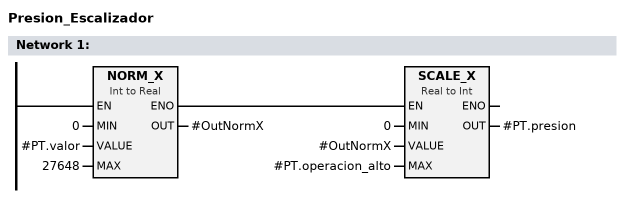
   RUNG wire#powerrail
      { S7_Templates := "[SrcType := Int, DestType := Real]"; S7_GenerateENO := "TRUE" } Normalize(min := 0, value := #PT.valor, max := 27648, out => #OutNormX)
      { S7_Templates := "[SrcType := Real, DestType := Int]"; S7_GenerateENO := "TRUE" } Scale(min := 0, value := #OutNormX, max := #PT.operacion_alto, out => #PT.presion)
   END_RUNG
   // the same network as SCL:
   // ENO of a box is taken as its EN; it also drops when the box reports an error
   #OutNormX := NORM_X(MIN := 0, VALUE := #PT.valor, MAX := 27648);
   #PT.presion := SCALE_X(MIN := 0, VALUE := #OutNormX, MAX := #PT.operacion_alto);
END_REGION
END_FUNCTION

FUNCTION "Nivel_RAD_Escalidar" : Void   // FC6, LAD
{ S7_Optimized_Access := 'TRUE' }
VERSION : 0.1
   VAR_IN_OUT
      RAD : "UDT_SENSORES_NIVEL";
   END_VAR
   VAR_TEMP
      OutNormX : Real;
      out : Int;
      Resultado_Transicion : Int;
      NivelAlto : Int;
      Resultado1 : Int;
      M1 : Real;
      M2 : Real;
   END_VAR
BEGIN

REGION Network 1
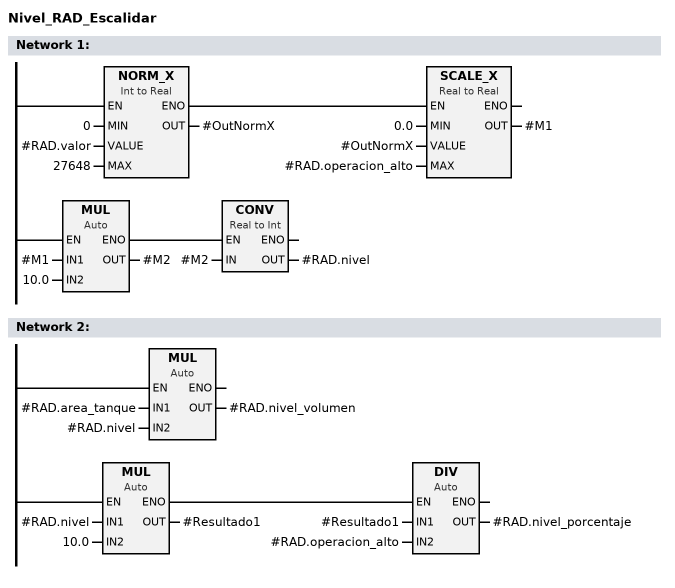
   RUNG wire#powerrail
      { S7_Templates := "[SrcType := Int, DestType := Real]"; S7_GenerateENO := "TRUE" } Normalize(min := 0, value := #RAD.valor, max := 27648, out => #OutNormX)
      { S7_Templates := "[SrcType := Real, DestType := Real]"; S7_GenerateENO := "TRUE" } Scale(min := 0.0, value := #OutNormX, max := #RAD.operacion_alto, out => #M1)
   END_RUNG
   RUNG wire#powerrail
      Mul(in1 := #M1, in2 := 10.0, out => #M2)
      { S7_Templates := "[SrcType := Real, DestType := Int]" } Convert(in := #M2, out => #RAD.nivel)
   END_RUNG
   // the same network as SCL:
   // ENO of a box is taken as its EN; it also drops when the box reports an error
   #OutNormX := NORM_X(MIN := 0, VALUE := #RAD.valor, MAX := 27648);
   #M1 := SCALE_X(MIN := 0.0, VALUE := #OutNormX, MAX := #RAD.operacion_alto);
   #M2 := #M1 * 10.0;
   #RAD.nivel := REAL_TO_INT(#M2);
END_REGION

REGION Network 2
   RUNG wire#powerrail
      Mul(in1 := #RAD.area_tanque, in2 := #RAD.nivel, out => #RAD.nivel_volumen)
   END_RUNG
   RUNG wire#powerrail
      Mul(in1 := #RAD.nivel, in2 := 10.0, out => #Resultado1)
      Div(in1 := #Resultado1, in2 := #RAD.operacion_alto, out => #RAD.nivel_porcentaje)
   END_RUNG
   // the same network as SCL:
   #RAD.nivel_volumen := #RAD.area_tanque * #RAD.nivel;
   #Resultado1 := #RAD.nivel * 10.0;
   #RAD.nivel_porcentaje := #Resultado1 / #RAD.operacion_alto;
END_REGION
END_FUNCTION

FUNCTION "Flujo_Escalizador" : Void   // FC7, LAD
{ S7_Optimized_Access := 'TRUE' }
VERSION : 0.1
   VAR_IN_OUT
      Flujo : "UDT_SENSORES_FLUJO";
   END_VAR
   VAR_TEMP
      OutNormX : Real;
      out : Int;
      Resultado_Transicion : Int;
   END_VAR
BEGIN

REGION Network 1
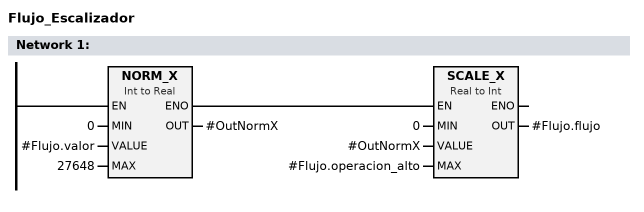
   RUNG wire#powerrail
      { S7_Templates := "[SrcType := Int, DestType := Real]"; S7_GenerateENO := "TRUE" } Normalize(min := 0, value := #Flujo.valor, max := 27648, out => #OutNormX)
      { S7_Templates := "[SrcType := Real, DestType := Int]"; S7_GenerateENO := "TRUE" } Scale(min := 0, value := #OutNormX, max := #Flujo.operacion_alto, out => #Flujo.flujo)
   END_RUNG
   // the same network as SCL:
   // ENO of a box is taken as its EN; it also drops when the box reports an error
   #OutNormX := NORM_X(MIN := 0, VALUE := #Flujo.valor, MAX := 27648);
   #Flujo.flujo := SCALE_X(MIN := 0, VALUE := #OutNormX, MAX := #Flujo.operacion_alto);
END_REGION
END_FUNCTION

ORGANIZATION_BLOCK "TransicionesINPUTOUTPUT"   // OB127, LAD, ProgramCycle
TITLE = "Main Program Sweep (Cycle)"
{ S7_Optimized_Access := 'TRUE' }
VERSION : 0.1
   VAR_INPUT
      Initial_Call : Bool;   // Initial call of this OB
      Remanence : Bool;   // =True, if remanent data are available
   END_VAR
   VAR_TEMP   // added for the SCL form of the ladder/FBD networks
      _w1 : Bool;
      _w2 : Bool;
      _w3 : Bool;
   END_VAR
BEGIN

REGION Network 1: BOMBA BC 11
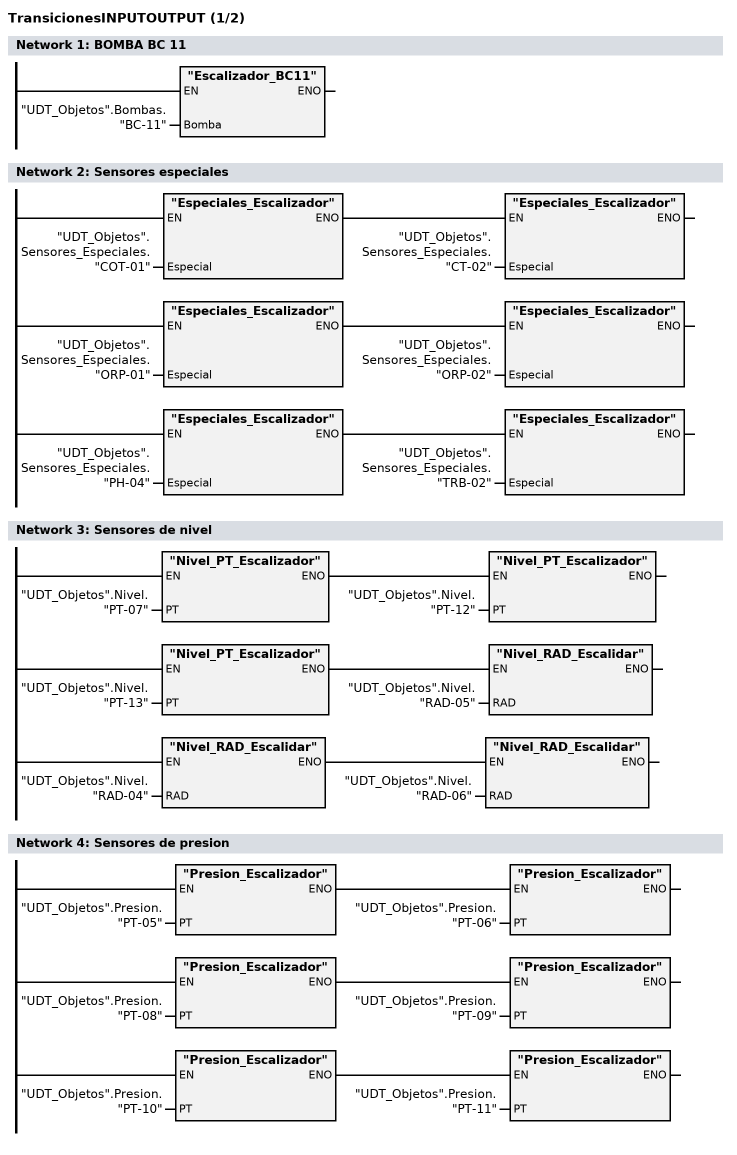
   RUNG wire#powerrail
      "Escalizador_BC11"(Bomba := "UDT_Objetos".Bombas."BC-11")
   END_RUNG
   // the same network as SCL:
   "Escalizador_BC11"(Bomba := "UDT_Objetos".Bombas."BC-11");
END_REGION

REGION Network 2: Sensores especiales
   RUNG wire#powerrail
      "Especiales_Escalizador"(Especial := "UDT_Objetos".Sensores_Especiales."COT-01")
      "Especiales_Escalizador"(Especial := "UDT_Objetos".Sensores_Especiales."CT-02")
   END_RUNG
   RUNG wire#powerrail
      "Especiales_Escalizador"(Especial := "UDT_Objetos".Sensores_Especiales."ORP-01")
      "Especiales_Escalizador"(Especial := "UDT_Objetos".Sensores_Especiales."ORP-02")
   END_RUNG
   RUNG wire#powerrail
      "Especiales_Escalizador"(Especial := "UDT_Objetos".Sensores_Especiales."PH-04")
      "Especiales_Escalizador"(Especial := "UDT_Objetos".Sensores_Especiales."TRB-02")
   END_RUNG
   // the same network as SCL:
   "Especiales_Escalizador"(Especial := "UDT_Objetos".Sensores_Especiales."COT-01", ENO => #_w1);
   IF #_w1 THEN "Especiales_Escalizador"(Especial := "UDT_Objetos".Sensores_Especiales."CT-02"); END_IF;
   "Especiales_Escalizador"(Especial := "UDT_Objetos".Sensores_Especiales."ORP-01", ENO => #_w2);
   IF #_w2 THEN "Especiales_Escalizador"(Especial := "UDT_Objetos".Sensores_Especiales."ORP-02"); END_IF;
   "Especiales_Escalizador"(Especial := "UDT_Objetos".Sensores_Especiales."PH-04", ENO => #_w3);
   IF #_w3 THEN "Especiales_Escalizador"(Especial := "UDT_Objetos".Sensores_Especiales."TRB-02"); END_IF;
END_REGION

REGION Network 3: Sensores de nivel
   RUNG wire#powerrail
      "Nivel_PT_Escalizador"(PT := "UDT_Objetos".Nivel."PT-07")
      "Nivel_PT_Escalizador"(PT := "UDT_Objetos".Nivel."PT-12")
   END_RUNG
   RUNG wire#powerrail
      "Nivel_PT_Escalizador"(PT := "UDT_Objetos".Nivel."PT-13")
      "Nivel_RAD_Escalidar"(RAD := "UDT_Objetos".Nivel."RAD-05")
   END_RUNG
   RUNG wire#powerrail
      "Nivel_RAD_Escalidar"(RAD := "UDT_Objetos".Nivel."RAD-04")
      "Nivel_RAD_Escalidar"(RAD := "UDT_Objetos".Nivel."RAD-06")
   END_RUNG
   // the same network as SCL:
   "Nivel_PT_Escalizador"(PT := "UDT_Objetos".Nivel."PT-07", ENO => #_w1);
   IF #_w1 THEN "Nivel_PT_Escalizador"(PT := "UDT_Objetos".Nivel."PT-12"); END_IF;
   "Nivel_PT_Escalizador"(PT := "UDT_Objetos".Nivel."PT-13", ENO => #_w2);
   IF #_w2 THEN "Nivel_RAD_Escalidar"(RAD := "UDT_Objetos".Nivel."RAD-05"); END_IF;
   "Nivel_RAD_Escalidar"(RAD := "UDT_Objetos".Nivel."RAD-04", ENO => #_w3);
   IF #_w3 THEN "Nivel_RAD_Escalidar"(RAD := "UDT_Objetos".Nivel."RAD-06"); END_IF;
END_REGION

REGION Network 4: Sensores de presion
   RUNG wire#powerrail
      "Presion_Escalizador"(PT := "UDT_Objetos".Presion."PT-05")
      "Presion_Escalizador"(PT := "UDT_Objetos".Presion."PT-06")
   END_RUNG
   RUNG wire#powerrail
      "Presion_Escalizador"(PT := "UDT_Objetos".Presion."PT-08")
      "Presion_Escalizador"(PT := "UDT_Objetos".Presion."PT-09")
   END_RUNG
   RUNG wire#powerrail
      "Presion_Escalizador"(PT := "UDT_Objetos".Presion."PT-10")
      "Presion_Escalizador"(PT := "UDT_Objetos".Presion."PT-11")
   END_RUNG
   // the same network as SCL:
   "Presion_Escalizador"(PT := "UDT_Objetos".Presion."PT-05", ENO => #_w1);
   IF #_w1 THEN "Presion_Escalizador"(PT := "UDT_Objetos".Presion."PT-06"); END_IF;
   "Presion_Escalizador"(PT := "UDT_Objetos".Presion."PT-08", ENO => #_w2);
   IF #_w2 THEN "Presion_Escalizador"(PT := "UDT_Objetos".Presion."PT-09"); END_IF;
   "Presion_Escalizador"(PT := "UDT_Objetos".Presion."PT-10", ENO => #_w3);
   IF #_w3 THEN "Presion_Escalizador"(PT := "UDT_Objetos".Presion."PT-11"); END_IF;
END_REGION

REGION Network 5
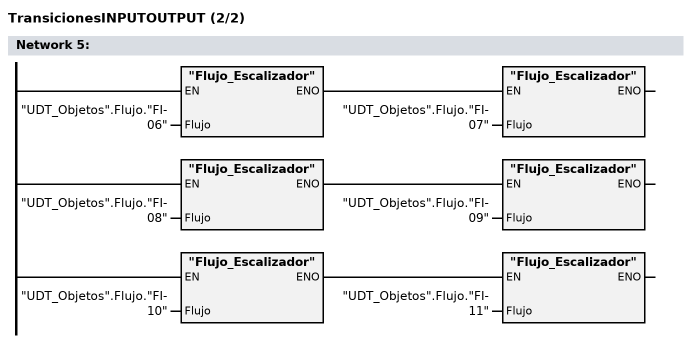
   RUNG wire#powerrail
      "Flujo_Escalizador"(Flujo := "UDT_Objetos".Flujo."FI-06")
      "Flujo_Escalizador"(Flujo := "UDT_Objetos".Flujo."FI-07")
   END_RUNG
   RUNG wire#powerrail
      "Flujo_Escalizador"(Flujo := "UDT_Objetos".Flujo."FI-08")
      "Flujo_Escalizador"(Flujo := "UDT_Objetos".Flujo."FI-09")
   END_RUNG
   RUNG wire#powerrail
      "Flujo_Escalizador"(Flujo := "UDT_Objetos".Flujo."FI-10")
      "Flujo_Escalizador"(Flujo := "UDT_Objetos".Flujo."FI-11")
   END_RUNG
   // the same network as SCL:
   "Flujo_Escalizador"(Flujo := "UDT_Objetos".Flujo."FI-06", ENO => #_w1);
   IF #_w1 THEN "Flujo_Escalizador"(Flujo := "UDT_Objetos".Flujo."FI-07"); END_IF;
   "Flujo_Escalizador"(Flujo := "UDT_Objetos".Flujo."FI-08", ENO => #_w2);
   IF #_w2 THEN "Flujo_Escalizador"(Flujo := "UDT_Objetos".Flujo."FI-09"); END_IF;
   "Flujo_Escalizador"(Flujo := "UDT_Objetos".Flujo."FI-10", ENO => #_w3);
   IF #_w3 THEN "Flujo_Escalizador"(Flujo := "UDT_Objetos".Flujo."FI-11"); END_IF;
END_REGION
END_ORGANIZATION_BLOCK

(* ===== HMI "HMI_RT_1" =====
system functions are stored by id; their names below are inferred from use
connection "HMI_Connection_1": ETHERNET, SMART_S7_1500_OMS

HMI tags "Default tag table"
   "UDT_Objetos_Bombas_BC-08_control" : Bool = PLC UDT_Objetos.Bombas.BC-08.control AT %DB1.DBX7182.0, 1 s
   "UDT_Objetos_Bombas_BC-09_control" : Bool = PLC UDT_Objetos.Bombas.BC-09.control AT %DB1.DBX7460.0, 1 s
   "UDT_Objetos_Bombas_BC-10_control" : Bool = PLC UDT_Objetos.Bombas.BC-10.control AT %DB1.DBX7738.0, 1 s
   "UDT_Objetos_Bombas_BC-11_control" : Bool = PLC UDT_Objetos.Bombas.BC-11.control AT %DB1.DBX8016.0, 1 s
   "UDT_Objetos_Bombas_BC-11_frecuencia" : Int = PLC UDT_Objetos.Bombas.BC-11.frecuencia AT %DB1.DBW8018, 1 s
   "UDT_Objetos_Bombas_BC-12_control" : Bool = PLC UDT_Objetos.Bombas.BC-12.control AT %DB1.DBX8294.0, 1 s
   "UDT_Objetos_Bombas_BC-13_control" : Bool = PLC UDT_Objetos.Bombas.BC-13.control AT %DB1.DBX8572.0, 1 s
   "UDT_Objetos_Dosificadoras_BD-AI-01_control" : Bool = PLC UDT_Objetos.Dosificadoras.BD-AI-01.control AT %DB1.DBX9938.0, 1 s
   "UDT_Objetos_Dosificadoras_BD-BIO-01_control" : Bool = PLC UDT_Objetos.Dosificadoras.BD-BIO-01.control AT %DB1.DBX10208.0, 1 s
   "UDT_Objetos_Bombas_BC-14_control" : Bool = PLC UDT_Objetos.Bombas.BC-14.control AT %DB1.DBX8850.0, 1 s
   "UDT_Objetos_Dosificadoras_BD-HIP-02_control" : Bool = PLC UDT_Objetos.Dosificadoras.BD-HIP-02.control AT %DB1.DBX10478.0, 1 s
   "UDT_Objetos_Dosificadoras_BD-HIP-01_control" : Bool = PLC UDT_Objetos.Dosificadoras.BD-HIP-01.control AT %DB1.DBX9128.0, 1 s
   "UDT_Objetos_Dosificadoras_BD-MBI-01_control" : Bool = PLC UDT_Objetos.Dosificadoras.BD-MBI-01.control AT %DB1.DBX9398.0, 1 s
   "UDT_Objetos_Dosificadoras_BD-UF-01_control" : Bool = PLC UDT_Objetos.Dosificadoras.BD-UF-01.control AT %DB1.DBX9668.0, 1 s
   "UDT_Objetos_Equipos_Especiales_BLW-01_control" : Bool = PLC UDT_Objetos.Equipos_Especiales.BLW-01.control AT %DB1.DBX25190.0, 1 s
   "UDT_Objetos_Equipos_Especiales_UV-01_control" : Bool = PLC UDT_Objetos.Equipos_Especiales.UV-01.control AT %DB1.DBX25458.0, 1 s
   "UDT_Objetos_Valvulas_VM-27_control" : Bool = PLC UDT_Objetos.Valvulas.VM-27.control AT %DB1.DBX0.0, 1 s
   "UDT_Objetos_Valvulas_VM-29_control" : Bool = PLC UDT_Objetos.Valvulas.VM-29.control AT %DB1.DBX266.0, 1 s
   "UDT_Objetos_Valvulas_VM-31_control" : Bool = PLC UDT_Objetos.Valvulas.VM-31.control AT %DB1.DBX532.0, 1 s
   "UDT_Objetos_Valvulas_VM-32_control" : Bool = PLC UDT_Objetos.Valvulas.VM-32.control AT %DB1.DBX798.0, 1 s
   "UDT_Objetos_Valvulas_VM-33_control" : Bool = PLC UDT_Objetos.Valvulas.VM-33.control AT %DB1.DBX1064.0, 1 s
   "UDT_Objetos_Valvulas_VM-34_control" : Bool = PLC UDT_Objetos.Valvulas.VM-34.control AT %DB1.DBX1330.0, 1 s
   "UDT_Objetos_Valvulas_VM-35_control" : Bool = PLC UDT_Objetos.Valvulas.VM-35.control AT %DB1.DBX1596.0, 1 s
   "UDT_Objetos_Valvulas_VM-36_control" : Bool = PLC UDT_Objetos.Valvulas.VM-36.control AT %DB1.DBX1862.0, 1 s
   "UDT_Objetos_Valvulas_VM-39_control" : Bool = PLC UDT_Objetos.Valvulas.VM-39.control AT %DB1.DBX2128.0, 1 s
   "UDT_Objetos_Valvulas_VM-40_control" : Bool = PLC UDT_Objetos.Valvulas.VM-40.control AT %DB1.DBX2394.0, 1 s
   "UDT_Objetos_Valvulas_VM-41_control" : Bool = PLC UDT_Objetos.Valvulas.VM-41.control AT %DB1.DBX2660.0, 1 s
   "UDT_Objetos_Valvulas_VM-42_control" : Bool = PLC UDT_Objetos.Valvulas.VM-42.control AT %DB1.DBX2926.0, 1 s
   "UDT_Objetos_Valvulas_VM-45_control" : Bool = PLC UDT_Objetos.Valvulas.VM-45.control AT %DB1.DBX3192.0, 1 s
   "UDT_Objetos_Valvulas_VM-46_control" : Bool = PLC UDT_Objetos.Valvulas.VM-46.control AT %DB1.DBX3458.0, 1 s
   "UDT_Objetos_Valvulas_VM-47_control" : Bool = PLC UDT_Objetos.Valvulas.VM-47.control AT %DB1.DBX3724.0, 1 s
   "UDT_Objetos_Valvulas_VM-48_control" : Bool = PLC UDT_Objetos.Valvulas.VM-48.control AT %DB1.DBX3990.0, 1 s
   "UDT_Objetos_Valvulas_VM-49_control" : Bool = PLC UDT_Objetos.Valvulas.VM-49.control AT %DB1.DBX4256.0, 1 s
   "UDT_Objetos_Valvulas_VM-50_control" : Bool = PLC UDT_Objetos.Valvulas.VM-50.control AT %DB1.DBX4522.0, 1 s
   "UDT_Objetos_Valvulas_VM-51_control" : Bool = PLC UDT_Objetos.Valvulas.VM-51.control AT %DB1.DBX4788.0, 1 s
   "UDT_Objetos_Valvulas_VM-52_control" : Bool = PLC UDT_Objetos.Valvulas.VM-52.control AT %DB1.DBX5054.0, 1 s
   "UDT_Objetos_Valvulas_VM-53_control" : Bool = PLC UDT_Objetos.Valvulas.VM-53.control AT %DB1.DBX5320.0, 1 s
   "UDT_Objetos_Valvulas_VM-56_control" : Bool = PLC UDT_Objetos.Valvulas.VM-56.control AT %DB1.DBX5586.0, 1 s
   "UDT_Objetos_Valvulas_VM-57_control" : Bool = PLC UDT_Objetos.Valvulas.VM-57.control AT %DB1.DBX5852.0, 1 s
   "UDT_Objetos_Valvulas_VM-58_control" : Bool = PLC UDT_Objetos.Valvulas.VM-58.control AT %DB1.DBX6118.0, 1 s
   "UDT_Objetos_Valvulas_VM-61_control" : Bool = PLC UDT_Objetos.Valvulas.VM-61.control AT %DB1.DBX6384.0, 1 s
   "UDT_Objetos_Valvulas_VM-62_control" : Bool = PLC UDT_Objetos.Valvulas.VM-62.control AT %DB1.DBX6650.0, 1 s
   "UDT_Objetos_Valvulas_VM-63_control" : Bool = PLC UDT_Objetos.Valvulas.VM-63.control AT %DB1.DBX6916.0, 1 s
   "UDT_Objetos_Valvulas_VM-27_estado" : Int = PLC UDT_Objetos.Valvulas.VM-27.estado AT %DB1.DBW2, 1 s
   "UDT_Objetos_Valvulas_VM-29_estado" : Int = PLC UDT_Objetos.Valvulas.VM-29.estado AT %DB1.DBW268, 1 s
   "UDT_Objetos_Valvulas_VM-31_estado" : Int = PLC UDT_Objetos.Valvulas.VM-31.estado AT %DB1.DBW534, 1 s
   "UDT_Objetos_Valvulas_VM-32_estado" : Int = PLC UDT_Objetos.Valvulas.VM-32.estado AT %DB1.DBW800, 1 s
   "UDT_Objetos_Valvulas_VM-33_estado" : Int = PLC UDT_Objetos.Valvulas.VM-33.estado AT %DB1.DBW1066, 1 s
   "UDT_Objetos_Valvulas_VM-34_estado" : Int = PLC UDT_Objetos.Valvulas.VM-34.estado AT %DB1.DBW1332, 1 s
   "UDT_Objetos_Valvulas_VM-35_estado" : Int = PLC UDT_Objetos.Valvulas.VM-35.estado AT %DB1.DBW1598, 1 s
   "UDT_Objetos_Valvulas_VM-36_estado" : Int = PLC UDT_Objetos.Valvulas.VM-36.estado AT %DB1.DBW1864, 1 s
   "UDT_Objetos_Valvulas_VM-39_estado" : Int = PLC UDT_Objetos.Valvulas.VM-39.estado AT %DB1.DBW2130, 1 s
   "UDT_Objetos_Valvulas_VM-40_estado" : Int = PLC UDT_Objetos.Valvulas.VM-40.estado AT %DB1.DBW2396, 1 s
   "UDT_Objetos_Valvulas_VM-41_estado" : Int = PLC UDT_Objetos.Valvulas.VM-41.estado AT %DB1.DBW2662, 1 s
   "UDT_Objetos_Valvulas_VM-42_estado" : Int = PLC UDT_Objetos.Valvulas.VM-42.estado AT %DB1.DBW2928, 1 s
   "UDT_Objetos_Valvulas_VM-45_estado" : Int = PLC UDT_Objetos.Valvulas.VM-45.estado AT %DB1.DBW3194, 1 s
   "UDT_Objetos_Valvulas_VM-46_estado" : Int = PLC UDT_Objetos.Valvulas.VM-46.estado AT %DB1.DBW3460, 1 s
   "UDT_Objetos_Valvulas_VM-47_estado" : Int = PLC UDT_Objetos.Valvulas.VM-47.estado AT %DB1.DBW3726, 1 s
   "UDT_Objetos_Valvulas_VM-48_estado" : Int = PLC UDT_Objetos.Valvulas.VM-48.estado AT %DB1.DBW3992, 1 s
   "UDT_Objetos_Valvulas_VM-49_estado" : Int = PLC UDT_Objetos.Valvulas.VM-49.estado AT %DB1.DBW4258, 1 s
   "UDT_Objetos_Valvulas_VM-50_estado" : Int = PLC UDT_Objetos.Valvulas.VM-50.estado AT %DB1.DBW4524, 1 s
   "UDT_Objetos_Valvulas_VM-51_estado" : Int = PLC UDT_Objetos.Valvulas.VM-51.estado AT %DB1.DBW4790, 1 s
   "UDT_Objetos_Valvulas_VM-52_estado" : Int = PLC UDT_Objetos.Valvulas.VM-52.estado AT %DB1.DBW5056, 1 s
   "UDT_Objetos_Valvulas_VM-53_estado" : Int = PLC UDT_Objetos.Valvulas.VM-53.estado AT %DB1.DBW5322, 1 s
   "UDT_Objetos_Valvulas_VM-56_estado" : Int = PLC UDT_Objetos.Valvulas.VM-56.estado AT %DB1.DBW5588, 1 s
   "UDT_Objetos_Valvulas_VM-57_estado" : Int = PLC UDT_Objetos.Valvulas.VM-57.estado AT %DB1.DBW5854, 1 s
   "UDT_Objetos_Valvulas_VM-58_estado" : Int = PLC UDT_Objetos.Valvulas.VM-58.estado AT %DB1.DBW6120, 1 s
   "UDT_Objetos_Valvulas_VM-61_estado" : Int = PLC UDT_Objetos.Valvulas.VM-61.estado AT %DB1.DBW6386, 1 s
   "UDT_Objetos_Valvulas_VM-62_estado" : Int = PLC UDT_Objetos.Valvulas.VM-62.estado AT %DB1.DBW6652, 1 s
   "UDT_Objetos_Valvulas_VM-63_estado" : Int = PLC UDT_Objetos.Valvulas.VM-63.estado AT %DB1.DBW6918, 1 s
   "UDT_Objetos_Bombas_BC-08_feedback" : Bool = PLC UDT_Objetos.Bombas.BC-08.feedback AT %DB1.DBX7186.0, 1 s
   "UDT_Objetos_Bombas_BC-08_estado" : Int = PLC UDT_Objetos.Bombas.BC-08.estado AT %DB1.DBW7192, 1 s
   "UDT_Objetos_Bombas_BC-09_estado" : Int = PLC UDT_Objetos.Bombas.BC-09.estado AT %DB1.DBW7470, 1 s
   "UDT_Objetos_Bombas_BC-10_estado" : Int = PLC UDT_Objetos.Bombas.BC-10.estado AT %DB1.DBW7748, 1 s
   "UDT_Objetos_Bombas_BC-11_estado" : Int = PLC UDT_Objetos.Bombas.BC-11.estado AT %DB1.DBW8026, 1 s
   "UDT_Objetos_Bombas_BC-12_estado" : Int = PLC UDT_Objetos.Bombas.BC-12.estado AT %DB1.DBW8304, 1 s
   "UDT_Objetos_Bombas_BC-13_estado" : Int = PLC UDT_Objetos.Bombas.BC-13.estado AT %DB1.DBW8582, 1 s
   "UDT_Objetos_Bombas_BC-14_estado" : Int = PLC UDT_Objetos.Bombas.BC-14.estado AT %DB1.DBW8860, 1 s
   "UDT_Objetos_Dosificadoras_BD-AI-01_estado" : Int = PLC UDT_Objetos.Dosificadoras.BD-AI-01.estado AT %DB1.DBW9940, 1 s
   "UDT_Objetos_Dosificadoras_BD-BIO-01_estado" : Int = PLC UDT_Objetos.Dosificadoras.BD-BIO-01.estado AT %DB1.DBW10210, 1 s
   "UDT_Objetos_Dosificadoras_BD-HIP-01_estado" : Int = PLC UDT_Objetos.Dosificadoras.BD-HIP-01.estado AT %DB1.DBW9130, 1 s
   "UDT_Objetos_Dosificadoras_BD-HIP-02_estado" : Int = PLC UDT_Objetos.Dosificadoras.BD-HIP-02.estado AT %DB1.DBW10480, 1 s
   "UDT_Objetos_Dosificadoras_BD-MBI-01_estado" : Int = PLC UDT_Objetos.Dosificadoras.BD-MBI-01.estado AT %DB1.DBW9400, 1 s
   "UDT_Objetos_Dosificadoras_BD-UF-01_estado" : Int = PLC UDT_Objetos.Dosificadoras.BD-UF-01.estado AT %DB1.DBW9670, 1 s
   "UDT_Objetos_Equipos_Especiales_BLW-01_estado" : Int = PLC UDT_Objetos.Equipos_Especiales.BLW-01.estado AT %DB1.DBW25194, 1 s
   "UDT_Objetos_Equipos_Especiales_UV-01_estado" : Int = PLC UDT_Objetos.Equipos_Especiales.UV-01.estado AT %DB1.DBW25462, 1 s
   "Solito" : Word = PLC Solito AT %MW2, 1 s
   "UDT_Objetos_Sensores_Especiales_COT-01_operacion_bajo" : Int = PLC UDT_Objetos.Sensores_Especiales.COT-01.operacion_bajo AT %DB1.DBW24920, 1 s
   "UDT_Objetos_Sensores_Especiales_COT-01_operacion_alto" : Int = PLC UDT_Objetos.Sensores_Especiales.COT-01.operacion_alto AT %DB1.DBW24918, 1 s
   "UDT_Objetos_Sensores_Especiales_COT-01_trabajo_alto" : Int = PLC UDT_Objetos.Sensores_Especiales.COT-01.trabajo_alto AT %DB1.DBW24924, 1 s
   "UDT_Objetos_Sensores_Especiales_CT-02_operacion_bajo" : Int = PLC UDT_Objetos.Sensores_Especiales.CT-02.operacion_bajo AT %DB1.DBW24390, 1 s
   "UDT_Objetos_Sensores_Especiales_CT-02_operacion_alto" : Int = PLC UDT_Objetos.Sensores_Especiales.CT-02.operacion_alto AT %DB1.DBW24388, 1 s
   "UDT_Objetos_Sensores_Especiales_CT-02_trabajo_alto" : Int = PLC UDT_Objetos.Sensores_Especiales.CT-02.trabajo_alto AT %DB1.DBW24394, 1 s
   "UDT_Objetos_Sensores_Especiales_CT-02_trabajo_bajo" : Int = PLC UDT_Objetos.Sensores_Especiales.CT-02.trabajo_bajo AT %DB1.DBW24396, 1 s
   "UDT_Objetos_Sensores_Especiales_ORP-01_operacion_bajo" : Int = PLC UDT_Objetos.Sensores_Especiales.ORP-01.operacion_bajo AT %DB1.DBW22800, 1 s
   "UDT_Objetos_Sensores_Especiales_ORP-01_operacion_alto" : Int = PLC UDT_Objetos.Sensores_Especiales.ORP-01.operacion_alto AT %DB1.DBW22798, 1 s
   "UDT_Objetos_Sensores_Especiales_ORP-01_trabajo_alto" : Int = PLC UDT_Objetos.Sensores_Especiales.ORP-01.trabajo_alto AT %DB1.DBW22804, 1 s
   "UDT_Objetos_Sensores_Especiales_ORP-01_trabajo_bajo" : Int = PLC UDT_Objetos.Sensores_Especiales.ORP-01.trabajo_bajo AT %DB1.DBW22806, 1 s
   "UDT_Objetos_Sensores_Especiales_ORP-02_operacion_bajo" : Int = PLC UDT_Objetos.Sensores_Especiales.ORP-02.operacion_bajo AT %DB1.DBW23330, 1 s
   "UDT_Objetos_Sensores_Especiales_ORP-02_operacion_alto" : Int = PLC UDT_Objetos.Sensores_Especiales.ORP-02.operacion_alto AT %DB1.DBW23328, 1 s
   "UDT_Objetos_Sensores_Especiales_ORP-02_trabajo_alto" : Int = PLC UDT_Objetos.Sensores_Especiales.ORP-02.trabajo_alto AT %DB1.DBW23334, 1 s
   "UDT_Objetos_Sensores_Especiales_ORP-02_trabajo_bajo" : Int = PLC UDT_Objetos.Sensores_Especiales.ORP-02.trabajo_bajo AT %DB1.DBW23336, 1 s
   "UDT_Objetos_Sensores_Especiales_PH-04_operacion_bajo" : Int = PLC UDT_Objetos.Sensores_Especiales.PH-04.operacion_bajo AT %DB1.DBW23860, 1 s
   "UDT_Objetos_Sensores_Especiales_TRB-02_operacion_bajo" : Int = PLC UDT_Objetos.Sensores_Especiales.TRB-02.operacion_bajo AT %DB1.DBW22270, 1 s
   "UDT_Objetos_Sensores_Especiales_TRB-02_operacion_alto" : Int = PLC UDT_Objetos.Sensores_Especiales.TRB-02.operacion_alto AT %DB1.DBW22268, 1 s
   "UDT_Objetos_Sensores_Especiales_TRB-02_trabajo_alto" : Int = PLC UDT_Objetos.Sensores_Especiales.TRB-02.trabajo_alto AT %DB1.DBW22274, 1 s
   "UDT_Objetos_Sensores_Especiales_TRB-02_trabajo_bajo" : Int = PLC UDT_Objetos.Sensores_Especiales.TRB-02.trabajo_bajo AT %DB1.DBW22276, 1 s
   "UDT_Objetos_Flujo_FI-06_operacion_bajo" : Int = PLC UDT_Objetos.Flujo.FI-06.operacion_bajo AT %DB1.DBW19330, 1 s
   "UDT_Objetos_Flujo_FI-06_operacion_alto" : Int = PLC UDT_Objetos.Flujo.FI-06.operacion_alto AT %DB1.DBW19328, 1 s
   "UDT_Objetos_Flujo_FI-06_trabajo_alto" : Int = PLC UDT_Objetos.Flujo.FI-06.trabajo_alto AT %DB1.DBW19332, 1 s
   "UDT_Objetos_Flujo_FI-06_trabajo_bajo" : Int = PLC UDT_Objetos.Flujo.FI-06.trabajo_bajo AT %DB1.DBW19334, 1 s
   "UDT_Objetos_Flujo_FI-07_operacion_bajo" : Int = PLC UDT_Objetos.Flujo.FI-07.operacion_bajo AT %DB1.DBW19864, 1 s
   "UDT_Objetos_Flujo_FI-07_operacion_alto" : Int = PLC UDT_Objetos.Flujo.FI-07.operacion_alto AT %DB1.DBW19862, 1 s
   "UDT_Objetos_Flujo_FI-07_trabajo_alto" : Int = PLC UDT_Objetos.Flujo.FI-07.trabajo_alto AT %DB1.DBW19866, 1 s
   "UDT_Objetos_Flujo_FI-07_trabajo_bajo" : Int = PLC UDT_Objetos.Flujo.FI-07.trabajo_bajo AT %DB1.DBW19868, 1 s
   "UDT_Objetos_Flujo_FI-08_operacion_bajo" : Int = PLC UDT_Objetos.Flujo.FI-08.operacion_bajo AT %DB1.DBW20398, 1 s
   "UDT_Objetos_Flujo_FI-08_operacion_alto" : Int = PLC UDT_Objetos.Flujo.FI-08.operacion_alto AT %DB1.DBW20396, 1 s
   "UDT_Objetos_Flujo_FI-08_trabajo_alto" : Int = PLC UDT_Objetos.Flujo.FI-08.trabajo_alto AT %DB1.DBW20400, 1 s
   "UDT_Objetos_Flujo_FI-08_trabajo_bajo" : Int = PLC UDT_Objetos.Flujo.FI-08.trabajo_bajo AT %DB1.DBW20402, 1 s
   "UDT_Objetos_Flujo_FI-09_operacion_bajo" : Int = PLC UDT_Objetos.Flujo.FI-09.operacion_bajo AT %DB1.DBW20932, 1 s
   "UDT_Objetos_Flujo_FI-09_operacion_alto" : Int = PLC UDT_Objetos.Flujo.FI-09.operacion_alto AT %DB1.DBW20930, 1 s
   "UDT_Objetos_Flujo_FI-09_trabajo_alto" : Int = PLC UDT_Objetos.Flujo.FI-09.trabajo_alto AT %DB1.DBW20934, 1 s
   "UDT_Objetos_Flujo_FI-09_trabajo_bajo" : Int = PLC UDT_Objetos.Flujo.FI-09.trabajo_bajo AT %DB1.DBW20936, 1 s
   "UDT_Objetos_Flujo_FI-11_operacion_alto" : Int = PLC UDT_Objetos.Flujo.FI-11.operacion_alto AT %DB1.DBW21998, 1 s
   "UDT_Objetos_Flujo_FI-11_trabajo_alto" : Int = PLC UDT_Objetos.Flujo.FI-11.trabajo_alto AT %DB1.DBW22002, 1 s
   "UDT_Objetos_Flujo_FI-11_trabajo_bajo" : Int = PLC UDT_Objetos.Flujo.FI-11.trabajo_bajo AT %DB1.DBW22004, 1 s
   "UDT_Objetos_Nivel_RAD-04_rango_alto" : Int = PLC UDT_Objetos.Nivel.RAD-04.operacion_alto AT %DB1.DBW11274, 1 s
   "UDT_Objetos_Nivel_RAD-05_rango_alto" : Int = PLC UDT_Objetos.Nivel.RAD-05.operacion_alto AT %DB1.DBW11816, 1 s
   "UDT_Objetos_Nivel_RAD-06_rango_alto" : Int = PLC UDT_Objetos.Nivel.RAD-06.operacion_alto AT %DB1.DBW12358, 1 s
   "UDT_Objetos_Nivel_RAD-04_rango_bajo" : Int = PLC UDT_Objetos.Nivel.RAD-04.rango_bajo AT %DB1.DBW11276, 1 s
   "UDT_Objetos_Nivel_RAD-04_rango_medio_bajo" : Int = PLC UDT_Objetos.Nivel.RAD-04.rango_medio_bajo AT %DB1.DBW11278, 1 s
   "UDT_Objetos_Nivel_RAD-04_rango_medio_alto" : Int = PLC UDT_Objetos.Nivel.RAD-04.rango_medio_alto AT %DB1.DBW11280, 1 s
   "UDT_Objetos_Nivel_RAD-04_rango_alto(1)" : Int = PLC UDT_Objetos.Nivel.RAD-04.rango_alto AT %DB1.DBW11282, 1 s
   "UDT_Objetos_Nivel_RAD-05_rango_bajo" : Int = PLC UDT_Objetos.Nivel.RAD-05.rango_bajo AT %DB1.DBW11818, 1 s
   "UDT_Objetos_Nivel_RAD-05_rango_medio_bajo" : Int = PLC UDT_Objetos.Nivel.RAD-05.rango_medio_bajo AT %DB1.DBW11820, 1 s
   "UDT_Objetos_Nivel_RAD-05_rango_medio_alto" : Int = PLC UDT_Objetos.Nivel.RAD-05.rango_medio_alto AT %DB1.DBW11822, 1 s
   "UDT_Objetos_Nivel_RAD-05_rango_alto(1)" : Int = PLC UDT_Objetos.Nivel.RAD-05.rango_alto AT %DB1.DBW11824, 1 s
   "UDT_Objetos_Nivel_RAD-06_rango_bajo" : Int = PLC UDT_Objetos.Nivel.RAD-06.rango_bajo AT %DB1.DBW12360, 1 s
   "UDT_Objetos_Nivel_RAD-06_rango_medio_bajo" : Int = PLC UDT_Objetos.Nivel.RAD-06.rango_medio_bajo AT %DB1.DBW12362, 1 s
   "UDT_Objetos_Nivel_RAD-06_rango_medio_alto" : Int = PLC UDT_Objetos.Nivel.RAD-06.rango_medio_alto AT %DB1.DBW12364, 1 s
   "UDT_Objetos_Nivel_RAD-06_rango_alto(1)" : Int = PLC UDT_Objetos.Nivel.RAD-06.rango_alto AT %DB1.DBW12366, 1 s
   "UDT_Objetos_Presion_PT-05_operacion_bajo" : Int = PLC UDT_Objetos.Presion.PT-05.operacion_bajo AT %DB1.DBW16148, 1 s
   "UDT_Objetos_Presion_PT-05_operacion_alto" : Int = PLC UDT_Objetos.Presion.PT-05.operacion_alto AT %DB1.DBW16146, 1 s
   "UDT_Objetos_Presion_PT-05_trabajo_bajo" : Int = PLC UDT_Objetos.Presion.PT-05.trabajo_bajo AT %DB1.DBW16152, 1 s
   "UDT_Objetos_Presion_PT-05_trabajo_alto" : Int = PLC UDT_Objetos.Presion.PT-05.trabajo_alto AT %DB1.DBW16150, 1 s
   "UDT_Objetos_Presion_PT-06_operacion_bajo" : Int = PLC UDT_Objetos.Presion.PT-06.operacion_bajo AT %DB1.DBW16678, 1 s
   "UDT_Objetos_Presion_PT-06_operacion_alto" : Int = PLC UDT_Objetos.Presion.PT-06.operacion_alto AT %DB1.DBW16676, 1 s
   "UDT_Objetos_Presion_PT-06_trabajo_bajo" : Int = PLC UDT_Objetos.Presion.PT-06.trabajo_bajo AT %DB1.DBW16682, 1 s
   "UDT_Objetos_Presion_PT-06_trabajo_alto" : Int = PLC UDT_Objetos.Presion.PT-06.trabajo_alto AT %DB1.DBW16680, 1 s
   "UDT_Objetos_Presion_PT-08_operacion_bajo" : Int = PLC UDT_Objetos.Presion.PT-08.operacion_bajo AT %DB1.DBW17208, 1 s
   "UDT_Objetos_Presion_PT-08_operacion_alto" : Int = PLC UDT_Objetos.Presion.PT-08.operacion_alto AT %DB1.DBW17206, 1 s
   "UDT_Objetos_Presion_PT-08_trabajo_bajo" : Int = PLC UDT_Objetos.Presion.PT-08.trabajo_bajo AT %DB1.DBW17212, 1 s
   "UDT_Objetos_Presion_PT-08_trabajo_alto" : Int = PLC UDT_Objetos.Presion.PT-08.trabajo_alto AT %DB1.DBW17210, 1 s
   "UDT_Objetos_Presion_PT-09_operacion_bajo" : Int = PLC UDT_Objetos.Presion.PT-09.operacion_bajo AT %DB1.DBW17738, 1 s
   "UDT_Objetos_Presion_PT-09_operacion_alto" : Int = PLC UDT_Objetos.Presion.PT-09.operacion_alto AT %DB1.DBW17736, 1 s
   "UDT_Objetos_Presion_PT-09_trabajo_bajo" : Int = PLC UDT_Objetos.Presion.PT-09.trabajo_bajo AT %DB1.DBW17742, 1 s
   "UDT_Objetos_Presion_PT-09_trabajo_alto" : Int = PLC UDT_Objetos.Presion.PT-09.trabajo_alto AT %DB1.DBW17740, 1 s
   "UDT_Objetos_Presion_PT-10_operacion_bajo" : Int = PLC UDT_Objetos.Presion.PT-10.operacion_bajo AT %DB1.DBW18268, 1 s
   "UDT_Objetos_Presion_PT-10_operacion_alto" : Int = PLC UDT_Objetos.Presion.PT-10.operacion_alto AT %DB1.DBW18266, 1 s
   "UDT_Objetos_Presion_PT-10_trabajo_bajo" : Int = PLC UDT_Objetos.Presion.PT-10.trabajo_bajo AT %DB1.DBW18272, 1 s
   "UDT_Objetos_Presion_PT-10_trabajo_alto" : Int = PLC UDT_Objetos.Presion.PT-10.trabajo_alto AT %DB1.DBW18270, 1 s
   "UDT_Objetos_Presion_PT-11_operacion_bajo" : Int = PLC UDT_Objetos.Presion.PT-11.operacion_bajo AT %DB1.DBW18798, 1 s
   "UDT_Objetos_Presion_PT-11_operacion_alto" : Int = PLC UDT_Objetos.Presion.PT-11.operacion_alto AT %DB1.DBW18796, 1 s
   "UDT_Objetos_Presion_PT-11_trabajo_bajo" : Int = PLC UDT_Objetos.Presion.PT-11.trabajo_bajo AT %DB1.DBW18802, 1 s
   "UDT_Objetos_Presion_PT-11_trabajo_alto" : Int = PLC UDT_Objetos.Presion.PT-11.trabajo_alto AT %DB1.DBW18800, 1 s
   "UDT_Objetos_Sensores_Especiales_COT-01_valor" : Int = PLC UDT_Objetos.Sensores_Especiales.COT-01.valor AT %DB1.DBW24660, 1 s
   "UDT_Objetos_Sensores_Especiales_CT-02_valor" : Int = PLC UDT_Objetos.Sensores_Especiales.CT-02.valor AT %DB1.DBW24130, 1 s
   "UDT_Objetos_Sensores_Especiales_ORP-01_valor" : Int = PLC UDT_Objetos.Sensores_Especiales.ORP-01.valor AT %DB1.DBW22540, 1 s
   "UDT_Objetos_Sensores_Especiales_ORP-02_valor" : Int = PLC UDT_Objetos.Sensores_Especiales.ORP-02.valor AT %DB1.DBW23070, 1 s
   "UDT_Objetos_Sensores_Especiales_PH-04_valor" : Int = PLC UDT_Objetos.Sensores_Especiales.PH-04.valor AT %DB1.DBW23600, 1 s
   "UDT_Objetos_Sensores_Especiales_TRB-02_valor" : Int = PLC UDT_Objetos.Sensores_Especiales.TRB-02.valor AT %DB1.DBW22010, 1 s
   "UDT_Objetos_Flujo_FI-06_valor" : Int = PLC UDT_Objetos.Flujo.FI-06.valor AT %DB1.DBW18806, 1 s
   "UDT_Objetos_Flujo_FI-07_valor" : Int = PLC UDT_Objetos.Flujo.FI-07.valor AT %DB1.DBW19340, 1 s
   "UDT_Objetos_Flujo_FI-08_valor" : Int = PLC UDT_Objetos.Flujo.FI-08.valor AT %DB1.DBW19874, 1 s
   "UDT_Objetos_Flujo_FI-09_valor" : Int = PLC UDT_Objetos.Flujo.FI-09.valor AT %DB1.DBW20408, 1 s
   "UDT_Objetos_Flujo_FI-10_valor" : Int = PLC UDT_Objetos.Flujo.FI-10.valor AT %DB1.DBW20942, 1 s
   "UDT_Objetos_Flujo_FI-11_valor" : Int = PLC UDT_Objetos.Flujo.FI-11.valor AT %DB1.DBW21476, 1 s
   "UDT_Objetos_Nivel_RAD-04_valor" : Int = PLC UDT_Objetos.Nivel.RAD-04.valor AT %DB1.DBW10748, 1 s
   "UDT_Objetos_Nivel_RAD-05_valor" : Int = PLC UDT_Objetos.Nivel.RAD-05.valor AT %DB1.DBW11290, 1 s
   "UDT_Objetos_Nivel_RAD-06_valor" : Int = PLC UDT_Objetos.Nivel.RAD-06.valor AT %DB1.DBW11832, 1 s
   "UDT_Objetos_Presion_PT-05_valor" : Int = PLC UDT_Objetos.Presion.PT-05.valor AT %DB1.DBW15626, 1 s
   "UDT_Objetos_Nivel_RAD-04_nivel" : Int = PLC UDT_Objetos.Nivel.RAD-04.nivel AT %DB1.DBW11006, 1 s
   "UDT_Objetos_Nivel_RAD-05_nivel" : Int = PLC UDT_Objetos.Nivel.RAD-05.nivel AT %DB1.DBW11548, 1 s
   "UDT_Objetos_Nivel_RAD-06_nivel" : Int = PLC UDT_Objetos.Nivel.RAD-06.nivel AT %DB1.DBW12090, 1 s
   "UDT_Objetos_Presion_PT-05_presion" : Int = PLC UDT_Objetos.Presion.PT-05.presion AT %DB1.DBW15884, 1 s
   "UDT_Objetos_Presion_PT-06_presion" : Int = PLC UDT_Objetos.Presion.PT-06.presion AT %DB1.DBW16414, 1 s
   "UDT_Objetos_Presion_PT-08_presion" : Int = PLC UDT_Objetos.Presion.PT-08.presion AT %DB1.DBW16944, 1 s
   "UDT_Objetos_Presion_PT-09_presion" : Int = PLC UDT_Objetos.Presion.PT-09.presion AT %DB1.DBW17474, 1 s
   "UDT_Objetos_Presion_PT-10_presion" : Int = PLC UDT_Objetos.Presion.PT-10.presion AT %DB1.DBW18004, 1 s
   "UDT_Objetos_Presion_PT-11_presion" : Int = PLC UDT_Objetos.Presion.PT-11.presion AT %DB1.DBW18534, 1 s
   "UDT_Objetos_Sensores_Especiales_COT-01_medicion" : Int = PLC UDT_Objetos.Sensores_Especiales.COT-01.medicion AT %DB1.DBW25188, 1 s
   "UDT_Objetos_Sensores_Especiales_CT-02_medicion" : Int = PLC UDT_Objetos.Sensores_Especiales.CT-02.medicion AT %DB1.DBW24658, 1 s
   "UDT_Objetos_Flujo_FI-06_flujo" : Int = PLC UDT_Objetos.Flujo.FI-06.flujo AT %DB1.DBW19338, 1 s
   "UDT_Objetos_Flujo_FI-07_flujo" : Int = PLC UDT_Objetos.Flujo.FI-07.flujo AT %DB1.DBW19872, 1 s
   "UDT_Objetos_Flujo_FI-08_flujo" : Int = PLC UDT_Objetos.Flujo.FI-08.flujo AT %DB1.DBW20406, 1 s
   "UDT_Objetos_Flujo_FI-09_flujo" : Int = PLC UDT_Objetos.Flujo.FI-09.flujo AT %DB1.DBW20940, 1 s
   "UDT_Objetos_Flujo_FI-10_flujo" : Int = PLC UDT_Objetos.Flujo.FI-10.flujo AT %DB1.DBW21474, 1 s
   "UDT_Objetos_Flujo_FI-11_flujo" : Int = PLC UDT_Objetos.Flujo.FI-11.flujo AT %DB1.DBW22008, 1 s
   "UDT_Objetos_Nivel_PT-07_nivel" : Int = PLC UDT_Objetos.Nivel.PT-07.nivel AT %DB1.DBW14258, 1 s
   "UDT_Objetos_Sensores_Especiales_ORP-01_medicion" : Int = PLC UDT_Objetos.Sensores_Especiales.ORP-01.medicion AT %DB1.DBW23068, 1 s
   "UDT_Objetos_Nivel_PT-12_nivel" : Int = PLC UDT_Objetos.Nivel.PT-12.nivel AT %DB1.DBW14800, 1 s
   "UDT_Objetos_Nivel_PT-13_nivel" : Int = PLC UDT_Objetos.Nivel.PT-13.nivel AT %DB1.DBW15342, 1 s
   "UDT_Objetos_Nivel_PT-07_rango_alto" : Int = PLC UDT_Objetos.Nivel.PT-07.rango_alto AT %DB1.DBW14534, 1 s
   "UDT_Objetos_Nivel_PT-07_rango_bajo" : Int = PLC UDT_Objetos.Nivel.PT-07.rango_bajo AT %DB1.DBW14528, 1 s
   "UDT_Objetos_Nivel_PT-07_rango_medio_bajo" : Int = PLC UDT_Objetos.Nivel.PT-07.rango_medio_bajo AT %DB1.DBW14530, 1 s
   "UDT_Objetos_Nivel_PT-07_operacion_alto" : Int = PLC UDT_Objetos.Nivel.PT-07.operacion_alto AT %DB1.DBW14526, 1 s
   "UDT_Objetos_Nivel_PT-07_rango_medio_alto" : Int = PLC UDT_Objetos.Nivel.PT-07.rango_medio_alto AT %DB1.DBW14532, 1 s
   "UDT_Objetos_Nivel_PT-12_operacion_alto" : Int = PLC UDT_Objetos.Nivel.PT-12.operacion_alto AT %DB1.DBW15068, 1 s
   "UDT_Objetos_Nivel_PT-12_rango_bajo" : Int = PLC UDT_Objetos.Nivel.PT-12.rango_bajo AT %DB1.DBW15070, 1 s
   "UDT_Objetos_Nivel_PT-12_rango_medio_bajo" : Int = PLC UDT_Objetos.Nivel.PT-12.rango_medio_bajo AT %DB1.DBW15072, 1 s
   "UDT_Objetos_Nivel_PT-12_rango_medio_alto" : Int = PLC UDT_Objetos.Nivel.PT-12.rango_medio_alto AT %DB1.DBW15074, 1 s
   "UDT_Objetos_Nivel_PT-12_rango_alto" : Int = PLC UDT_Objetos.Nivel.PT-12.rango_alto AT %DB1.DBW15076, 1 s
   "UDT_Objetos_Nivel_PT-13_operacion_alto" : Int = PLC UDT_Objetos.Nivel.PT-13.operacion_alto AT %DB1.DBW15610, 1 s
   "UDT_Objetos_Nivel_PT-13_rango_bajo" : Int = PLC UDT_Objetos.Nivel.PT-13.rango_bajo AT %DB1.DBW15612, 1 s
   "UDT_Objetos_Nivel_PT-13_rango_medio_bajo" : Int = PLC UDT_Objetos.Nivel.PT-13.rango_medio_bajo AT %DB1.DBW15614, 1 s
   "UDT_Objetos_Nivel_PT-13_rango_medio_alto" : Int = PLC UDT_Objetos.Nivel.PT-13.rango_medio_alto AT %DB1.DBW15616, 1 s
   "UDT_Objetos_Nivel_PT-13_rango_alto" : Int = PLC UDT_Objetos.Nivel.PT-13.rango_alto AT %DB1.DBW15618, 1 s
   "UDT_Objetos_Nivel_RAD-04_area_tanque" : Int = PLC UDT_Objetos.Nivel.RAD-04.area_tanque AT %DB1.DBW11284, 1 s
   "UDT_Objetos_Nivel_PT-12_area_tanque" : Int = PLC UDT_Objetos.Nivel.PT-12.area_tanque AT %DB1.DBW15078, 1 s
   "UDT_Objetos_Nivel_PT-13_area_tanque" : Int = PLC UDT_Objetos.Nivel.PT-13.area_tanque AT %DB1.DBW15620, 1 s
   "UDT_Objetos_Nivel_PT-07_area_tanque" : Int = PLC UDT_Objetos.Nivel.PT-07.area_tanque AT %DB1.DBW14536, 1 s
   "UDT_Objetos_Nivel_RAD-05_area_tanque" : Int = PLC UDT_Objetos.Nivel.RAD-05.area_tanque AT %DB1.DBW11826, 1 s
   "UDT_Objetos_Nivel_RAD-06_area_tanque" : Int = PLC UDT_Objetos.Nivel.RAD-06.area_tanque AT %DB1.DBW12368, 1 s
   "UDT_Objetos_Nivel_RAD-04_nivel_porcentaje" : Int = PLC UDT_Objetos.Nivel.RAD-04.nivel_porcentaje AT %DB1.DBW11286, 1 s
   "UDT_Objetos_Nivel_PT-13_nivel_porcentaje" : Int = PLC UDT_Objetos.Nivel.PT-13.nivel_porcentaje AT %DB1.DBW15622, 1 s
   "UDT_Objetos_Nivel_RAD-04_nivel_volumen" : Int = PLC UDT_Objetos.Nivel.RAD-04.nivel_volumen AT %DB1.DBW11288, 1 s
   "UDT_Objetos_Nivel_PT-07_nivel_porcentaje" : Int = PLC UDT_Objetos.Nivel.PT-07.nivel_porcentaje AT %DB1.DBW14538, 1 s
   "UDT_Objetos_Nivel_PT-07_nivel_volumen" : Int = PLC UDT_Objetos.Nivel.PT-07.nivel_volumen AT %DB1.DBW14540, 1 s
   "UDT_Objetos_Nivel_PT-12_nivel_porcentaje" : Int = PLC UDT_Objetos.Nivel.PT-12.nivel_porcentaje AT %DB1.DBW15080, 1 s
   "UDT_Objetos_Nivel_PT-12_nivel_volumen" : Int = PLC UDT_Objetos.Nivel.PT-12.nivel_volumen AT %DB1.DBW15082, 1 s
   "UDT_Objetos_Nivel_RAD-06_nivel_volumen" : Int = PLC UDT_Objetos.Nivel.RAD-06.nivel_volumen AT %DB1.DBW12372, 1 s
   "UDT_Objetos_Nivel_RAD-06_nivel_porcentaje" : Int = PLC UDT_Objetos.Nivel.RAD-06.nivel_porcentaje AT %DB1.DBW12370, 1 s
   "UDT_Objetos_Nivel_RAD-05_nivel_volumen" : Int = PLC UDT_Objetos.Nivel.RAD-05.nivel_volumen AT %DB1.DBW11830, 1 s
   "UDT_Objetos_Nivel_RAD-05_nivel_porcentaje" : Int = PLC UDT_Objetos.Nivel.RAD-05.nivel_porcentaje AT %DB1.DBW11828, 1 s
   "UDT_Objetos_Nivel_PT-13_nivel_volumen" : Int = PLC UDT_Objetos.Nivel.PT-13.nivel_volumen AT %DB1.DBW15624, 1 s
   "UDT_Objetos_AlarmasTotales_AlarmasBombas" : Int = PLC UDT_Objetos.AlarmasTotales.AlarmasBombas AT %DB1.DBW25750, 1 s
   "UDT_Objetos_AlarmasTotales_AlarmasDosificadoras" : Int = PLC UDT_Objetos.AlarmasTotales.AlarmasDosificadoras AT %DB1.DBW25748, 1 s
   "UDT_Objetos_AlarmasTotales_AlarmasEspeciales" : Int = PLC UDT_Objetos.AlarmasTotales.AlarmasEspeciales AT %DB1.DBW25746, 1 s
   "UDT_Objetos_AlarmasTotales_AlarmasFlujo" : Int = PLC UDT_Objetos.AlarmasTotales.AlarmasFlujo AT %DB1.DBW25752, 1 s
   "UDT_Objetos_AlarmasTotales_AlarmasTanques" : Int = PLC UDT_Objetos.AlarmasTotales.AlarmasTanques AT %DB1.DBW25754, 1 s
   "UDT_Objetos_AlarmasTotales_AlarmasPresion" : Int = PLC UDT_Objetos.AlarmasTotales.AlarmasPresion AT %DB1.DBW25744, 1 s
   "UDT_Objetos_AlarmasTotales_AlarmasValvulas1" : Int, internal
   "UDT_Objetos_AlarmasTotales_AlarmasValvulas2" : Int = PLC UDT_Objetos.AlarmasTotales.AlarmasValvulas2 AT %DB1.DBW25742, 1 s
   "UDT_Objetos_ProcesoUF_ProcessName" : String[20] = PLC UDT_Objetos.ProcesoUF.ProcessName AT %DB1.DBX25758.0, 1 s
   "UDT_Objetos_Bombas_BC-11_alarma" : Bool = PLC UDT_Objetos.Bombas.BC-11.alarma AT %DB1.DBX8028.0, 1 s

HMI tags "Adicionales"
   "M1" : Bool, internal
   "PantallaActual" : Real, internal
   "Probando alarmas" : Real, internal

discrete alarms
   1: 'Falla BC-08', class UF, trigger "UDT_Objetos_AlarmasTotales_AlarmasBombas" bit 0
   2: 'Falla BC-09', class UF, trigger "UDT_Objetos_AlarmasTotales_AlarmasBombas" bit 1
   3: 'Falla BC-10', class UF, trigger "UDT_Objetos_AlarmasTotales_AlarmasBombas" bit 2
   4: 'Frecuencia baja, bomba BC-11', class OI, trigger "UDT_Objetos_AlarmasTotales_AlarmasBombas" bit 3
   5: 'Falla BC-12', class OI, trigger "UDT_Objetos_AlarmasTotales_AlarmasBombas" bit 4
   6: 'Falla BC-13', class PER, trigger "UDT_Objetos_AlarmasTotales_AlarmasBombas" bit 5
   7: 'Falla BC-14', class RECH, trigger "UDT_Objetos_AlarmasTotales_AlarmasBombas" bit 6
   8: 'Falla BD-UF-01', class UF, trigger "UDT_Objetos_AlarmasTotales_AlarmasDosificadoras" bit 0
   9: 'Falla BD-AI-01', class OI, trigger "UDT_Objetos_AlarmasTotales_AlarmasDosificadoras" bit 1
   10: 'Falla BD-HIP-01', class UF, trigger "UDT_Objetos_AlarmasTotales_AlarmasDosificadoras" bit 2
   11: 'Falla BD-HIP-02', class PER, trigger "UDT_Objetos_AlarmasTotales_AlarmasDosificadoras" bit 3
   12: 'Falla BD-BIO-01', class OI, trigger "UDT_Objetos_AlarmasTotales_AlarmasDosificadoras" bit 4
   13: 'Falla BD-MBI-01', class UF, trigger "UDT_Objetos_AlarmasTotales_AlarmasDosificadoras" bit 5
   14: 'Falla BLW-01', class UF bit 0
   15: 'Falla UV-01', class PER bit 0
   16: 'Falla COT-01', class PER, trigger "UDT_Objetos_AlarmasTotales_AlarmasEspeciales" bit 0
   17: 'COT alto, Salida TK-PER-01', class PER, trigger "UDT_Objetos_AlarmasTotales_AlarmasEspeciales" bit 1
   18: 'Automático PER suspendido, COT alto', class PER, trigger "UDT_Objetos_AlarmasTotales_AlarmasEspeciales" bit 2
   19: 'Falla CT-02', class OI, trigger "UDT_Objetos_AlarmasTotales_AlarmasEspeciales" bit 3
   20: 'Conductividad fuera del rango superior, permeado osmosis', class OI, trigger "UDT_Objetos_AlarmasTotales_AlarmasEspeciales" bit 4
   21: 'Conductividad fuera del rango inferior, permeado osmosis', class OI, trigger "UDT_Objetos_AlarmasTotales_AlarmasEspeciales" bit 5
   22: 'Falla ORP-01', class OI, trigger "UDT_Objetos_AlarmasTotales_AlarmasEspeciales" bit 6
   23: 'ORP alto, entrada osmosis', class OI, trigger "UDT_Objetos_AlarmasTotales_AlarmasEspeciales" bit 7
   24: 'Falla ORP-02', class PER, trigger "UDT_Objetos_AlarmasTotales_AlarmasEspeciales" bit 8
   25: 'ORP alto, Salida tanque 5', class PER, trigger "UDT_Objetos_AlarmasTotales_AlarmasEspeciales" bit 9
   26: 'ORP bajo, Salida 1', class PER, trigger "UDT_Objetos_AlarmasTotales_AlarmasEspeciales" bit 10
   27: 'Permeado tanque 5, suspendido ORP alto', class PER, trigger "UDT_Objetos_AlarmasTotales_AlarmasEspeciales" bit 11
   28: 'Falla PH-04', class OI, trigger "UDT_Objetos_AlarmasTotales_AlarmasEspeciales" bit 12
   29: 'Falla TRB-02', class UF, trigger "UDT_Objetos_AlarmasTotales_AlarmasEspeciales" bit 13
   30: 'NTU fuera del rango superior salida UF', class UF, trigger "UDT_Objetos_AlarmasTotales_AlarmasEspeciales" bit 14
   31: 'NTU fuera del rango inferior salida UF', class UF, trigger "UDT_Objetos_AlarmasTotales_AlarmasEspeciales" bit 15
   32: 'Caudal fuera del rango superior, entrada UF', class UF, trigger "UDT_Objetos_AlarmasTotales_AlarmasFlujo" bit 0
   33: 'Caudal fuera del rango inferior, entrada UF', class UF, trigger "UDT_Objetos_AlarmasTotales_AlarmasFlujo" bit 1
   34: 'Caudal fuera del rango superior, salida UF', class UF, trigger "UDT_Objetos_AlarmasTotales_AlarmasFlujo" bit 2
   35: 'Caudal fuera del rango inferior, salida UF', class UF, trigger "UDT_Objetos_AlarmasTotales_AlarmasFlujo" bit 3
   36: 'Caudal fuera del rango superior, entrada osmosis', class OI, trigger "UDT_Objetos_AlarmasTotales_AlarmasFlujo" bit 4
   37: 'Caudal fuera del rango inferior, entrada osmosis', class OI, trigger "UDT_Objetos_AlarmasTotales_AlarmasFlujo" bit 5
   38: 'Caudal fuera del rango superior, permeado osmosis', class OI, trigger "UDT_Objetos_AlarmasTotales_AlarmasFlujo" bit 6
   39: 'Caudal fuera del rango inferior, permeado osmosis', class OI, trigger "UDT_Objetos_AlarmasTotales_AlarmasFlujo" bit 7
   40: 'Caudal fuera del rango superior, rechazo osmosis', class OI, trigger "UDT_Objetos_AlarmasTotales_AlarmasFlujo" bit 8
   41: 'Caudal fuera del rango inferior, rechazo osmosis', class OI, trigger "UDT_Objetos_AlarmasTotales_AlarmasFlujo" bit 9
   42: 'Nivel bajo TK-CIP', class OI, trigger "UDT_Objetos_AlarmasTotales_AlarmasTanques" bit 0
   43: 'Nivel bajo TK-AI-01', class OI, trigger "UDT_Objetos_AlarmasTotales_AlarmasTanques" bit 1
   44: 'Nivel bajo TK-BIO-01', class OI, trigger "UDT_Objetos_AlarmasTotales_AlarmasTanques" bit 2
   45: 'Nivel bajo TK-HIP-01', class UF, trigger "UDT_Objetos_AlarmasTotales_AlarmasTanques" bit 3
   46: 'Nivel bajo TK-HIP-02', class PER, trigger "UDT_Objetos_AlarmasTotales_AlarmasTanques" bit 4
   47: 'Nivel bajo TK-MBI-01', class UF, trigger "UDT_Objetos_AlarmasTotales_AlarmasTanques" bit 5
   48: 'Nivel bajo TK-UF-02', class UF, trigger "UDT_Objetos_AlarmasTotales_AlarmasTanques" bit 6
   49: 'Nivel alto, linea de permeado 1', class RECH, trigger "UDT_Objetos_AlarmasTotales_AlarmasTanques" bit 7
   50: 'Tanque cisterna TK-06, lleno', class UF, trigger "UDT_Objetos_AlarmasTotales_AlarmasTanques" bit 8
   51: 'Tanque 4, lleno', class PER, trigger "UDT_Objetos_AlarmasTotales_AlarmasTanques" bit 9
   52: 'Tanque 5, lleno', class PER, trigger "UDT_Objetos_AlarmasTotales_AlarmasTanques" bit 10
   53: 'Presión baja, entrada UF', class UF, trigger "UDT_Objetos_AlarmasTotales_AlarmasPresion" bit 0
   54: 'Presión alta, entrada UF', class UF, trigger "UDT_Objetos_AlarmasTotales_AlarmasPresion" bit 1
   55: 'Presión baja, salida UF', class UF, trigger "UDT_Objetos_AlarmasTotales_AlarmasPresion" bit 2
   56: 'Presión alta, salida UF', class UF, trigger "UDT_Objetos_AlarmasTotales_AlarmasPresion" bit 3
   57: 'Tanque TK-UF-01, lleno', class UF, trigger "UDT_Objetos_AlarmasTotales_AlarmasTanques" bit 11
   58: 'Tanque TK-UF-01, lleno', class UF, trigger "UDT_Objetos_AlarmasTotales_AlarmasTanques" bit 12
   59: 'Presión baja, entrada osmosis', class OI, trigger "UDT_Objetos_AlarmasTotales_AlarmasPresion" bit 4
   60: 'Presión baja, sistema de osmosis', class OI, trigger "UDT_Objetos_AlarmasTotales_AlarmasPresion" bit 5
   61: 'Presión alta, sistema de osmosis', class OI, trigger "UDT_Objetos_AlarmasTotales_AlarmasPresion" bit 6
   62: 'Sistema de osmosis, requiere CIP', class OI, trigger "UDT_Objetos_AlarmasTotales_AlarmasPresion" bit 7
   63: 'Tanque TK-PER-01, lleno', class PER, trigger "UDT_Objetos_AlarmasTotales_AlarmasTanques" bit 13
   64: 'Tanque TK-PER-01, lleno', class PER, trigger "UDT_Objetos_AlarmasTotales_AlarmasTanques" bit 14
   65: 'Tanque rechazo OI, lleno', class RECH, trigger "UDT_Objetos_AlarmasTotales_AlarmasTanques" bit 15
   66: 'Válvula VM-29, Salida tanque 6 a UF no abre', class UF, trigger "UDT_Objetos_AlarmasTotales_AlarmasValvulas1" bit 0
   67: 'Válvula VM-31, Entrada UF no abre', class UF, trigger "UDT_Objetos_AlarmasTotales_AlarmasValvulas1" bit 1
   68: 'Válvula VM-31, Entrada UF, no cierra', class UF, trigger "UDT_Objetos_AlarmasTotales_AlarmasValvulas1" bit 2
   69: 'Válvula VM-32, Salida BLW-01, no abre', class UF, trigger "UDT_Objetos_AlarmasTotales_AlarmasValvulas1" bit 3
   70: 'Válvula VM-33, Desague inferior UF, no abre', class UF, trigger "UDT_Objetos_AlarmasTotales_AlarmasValvulas1" bit 4
   71: 'Válvula VM-34, Desague superior UF, no abre', class UF, trigger "UDT_Objetos_AlarmasTotales_AlarmasValvulas1" bit 5
   72: 'Válvula VM-35, Desague superior UF tanque TK-UF-01, no abre', class UF, trigger "UDT_Objetos_AlarmasTotales_AlarmasValvulas1" bit 6
   73: 'Válvula VM-36, Salida UF, no abre', class UF, trigger "UDT_Objetos_AlarmasTotales_AlarmasValvulas1" bit 7
   74: 'Válvula VM-39, Descarga BC-09 UF, no abre', class UF, trigger "UDT_Objetos_AlarmasTotales_AlarmasValvulas1" bit 8
   75: 'Válvula VM-40, Salida UF, no abre', class UF, trigger "UDT_Objetos_AlarmasTotales_AlarmasValvulas1" bit 9
   76: 'Válvula VM-41, Salida UF, no abre', class UF, trigger "UDT_Objetos_AlarmasTotales_AlarmasValvulas1" bit 10
   77: 'Válvula VM-42, Purga TK-UF-01, no abre', class UF, trigger "UDT_Objetos_AlarmasTotales_AlarmasValvulas1" bit 11
   78: 'Válvula VM-42, Purga TK-UF-01, no cierra', class UF, trigger "UDT_Objetos_AlarmasTotales_AlarmasValvulas1" bit 12
   79: 'Válvula VM-45, entrada osmosis bomba BC-10 no abre', class OI, trigger "UDT_Objetos_AlarmasTotales_AlarmasValvulas1" bit 13
   80: 'Válvula VM-46, by-pass bomba BC-10 no abre', class OI, trigger "UDT_Objetos_AlarmasTotales_AlarmasValvulas1" bit 14
   81: 'Válvula VM-47, descarga bomba BC-11 no abre', class OI, trigger "UDT_Objetos_AlarmasTotales_AlarmasValvulas1" bit 15
   82: 'Válvula VM-48, descarga bomba BC-10 no abre', class OI, trigger "UDT_Objetos_AlarmasTotales_AlarmasValvulas2" bit 0
   83: 'Válvula VM-49, entrada permeado TK-CIP, no abre', class OI, trigger "UDT_Objetos_AlarmasTotales_AlarmasValvulas2" bit 1
   84: 'Válvula VM-49, entrada permeado TK-CIP, no cierra', class OI, trigger "UDT_Objetos_AlarmasTotales_AlarmasValvulas2" bit 2
   85: 'Válvula VM-50, entrada rechazo TK-CIP, no cierra', class OI, trigger "UDT_Objetos_AlarmasTotales_AlarmasValvulas2" bit 3
   86: 'Válvula VM-51, entrada agua limpia TK-CIP, no abre', class OI, trigger "UDT_Objetos_AlarmasTotales_AlarmasValvulas2" bit 4
   87: 'Válvula VM-51, entrada agua limpia TK-CIP, no cierra', class OI, trigger "UDT_Objetos_AlarmasTotales_AlarmasValvulas2" bit 5
   88: 'Válvula VM-52, rechazo osmosis, no abre', class OI, trigger "UDT_Objetos_AlarmasTotales_AlarmasValvulas2" bit 6
   89: 'Válvula VM-52, Purga TK-CIP, no abre', class OI, trigger "UDT_Objetos_AlarmasTotales_AlarmasValvulas2" bit 7
   90: 'Válvula VM-52, Purga TK-CIP, no cierra', class OI, trigger "UDT_Objetos_AlarmasTotales_AlarmasValvulas2" bit 8
   91: 'Válvula VM-56, permeado osmosis, no abre', class OI, trigger "UDT_Objetos_AlarmasTotales_AlarmasValvulas2" bit 9
   92: 'Válvula VM-57, permeado osmosis, no abre', class OI, trigger "UDT_Objetos_AlarmasTotales_AlarmasValvulas2" bit 10
   93: 'Válvula VM-58, Purga TK-PER-01, no abre', class PER, trigger "UDT_Objetos_AlarmasTotales_AlarmasValvulas2" bit 11
   94: 'Válvula VM-58, Purga TK-PER-01, no cierra', class PER, trigger "UDT_Objetos_AlarmasTotales_AlarmasValvulas2" bit 12
   95: 'Válvula VM-61, permeado tanque 5, no abre', class PER, trigger "UDT_Objetos_AlarmasTotales_AlarmasValvulas2" bit 13
   96: 'Válvula VM-62, permeado tanque 4, no abre', class PER, trigger "UDT_Objetos_AlarmasTotales_AlarmasValvulas2" bit 14
   97: 'Válvula VM-63, CIP-TPER, no abre', class PER, trigger "UDT_Objetos_AlarmasTotales_AlarmasValvulas2" bit 15

graphic list "Valvulas": 0 'valvulaOff'; 1 'valvulaOn'; 2 'valvulaFalla'

graphic list "Bombas": 0 'bombaOff'; 1 'bombaOn'; 2 'bombaFalla'

graphic list "Blower": 0 'blowerOff'; 1 'blowerOn'; 2 'blowerFalla'

graphic list "ValvulasRotadas": 0 'valvulaOffRotate_1'; 1 'valvulaOnRotate_1'; 2 'valvulaFallaRotate_1'

graphic list "Dosificadoras": 0 'dosificadoraOff'; 1 'dosificadoraOn'; 2 'dosificadoraFalla'

graphic list "BombaDerechas": 0 'bombaOffDerecha'; 1 'bombaOnDerecha'; 2 'bombaFallaDerecha'

graphic list "BombasIzquierdas": 0 'bombaOffIzquierda'; 1 'bombaOnIzquierda'; 2 'bombaFallaIzquierda'

graphic list "DosificadorasIzquierdas": 0 'dosificadoraOffIzquierda'; 1 'dosificadoraOnIzquierda'; 2 'dosificadoraFallaIzquierda'

graphic list "DosificadorasDerecha": 0 'disificadorOffDerecha'; 1 'disificadorOnDerecha'; 2 'disificadorFallaDerecha'

graphic list "BombaGrande": 0 'bombaGrandeOff'; 1 'bombaGrandeOn'; 2 'bombaGrandeFalla'

graphic list "Ultravioleta": 0 'ultravioletaOff'; 1 'ultravioletaOn'; 2 'ultravioletaFalla'

Template "Template_1" 800x480
   Button "Template_Button_3" at 400,440 size 100x39; TextOff 'MANUAL'
      on Click: ActivateScreen("Manual", 0)
   Button "Template_Button_4" at 300,440 size 100x39; TextOff 'GRAFICAS'
      on Click: ActivateScreen("COT", 0)
   Button "Template_Button_5" at 200,440 size 100x39; TextOff 'PRODUCCION PER'
      on Click: ActivateScreen("Produccion PER", 0)
   Button "Template_Button_6" at 100,440 size 100x39; TextOff 'PRODUCCION OI'
      on Click: ActivateScreen("Produccion OI", 0)
   Button "Template_Button_7" at 0,440 size 100x39; TextOff 'PRODUCCION UF'
      on Click: ActivateScreen("Produccion UF", 0)
   Button "Template_Button_9" at 500,440 size 99x39; TextOff 'INICIO'
      on Click: ActivateScreen("0Ultrafiltracion", 0)
   Group "Group" at 300,62 size 200x24
   TextField "Template_Text field_1" at 300,62 size 61x24; Text 'Proceso'
   IOField "Template_I/O field_1" at 359,62 size 141x24; FormatPattern ??????????
      ProcessValue <- "UDT_Objetos_ProcesoUF_ProcessName"

screen "0Ultrafiltracion" 800x480, template "Template_1"
   on GenerateScreen: SetTag("PantallaActual", 1)
   Button "Button_1" at 694,0 size 106x56; TextOff 'AJUSTES'
      on Click: ActivateScreen("Configuraciones", 0)
   AlarmView "Alarm view_1" at 111,0 size 584x56
      on Activate: ActivateScreen("Alarmas", 0)
   GraphicView "Graphic view_1" at 0,0 size 112x56; Picture "Coca-Cola_Femsa_Logo"
   GraphicView "Graphic view_2" at 0,107 size 800x332; Picture "ULTRAFICAION_4"
   GraphicIOField "Graphic I/O field_1" at 36,181 size 30x30; PictureList "Valvulas"
      ProcessValue <- "UDT_Objetos_Valvulas_VM-27_estado"
   GraphicIOField "Graphic I/O field_2" at 160,272 size 30x30; PictureList "Valvulas"
      ProcessValue <- "UDT_Objetos_Valvulas_VM-29_estado"
   GraphicIOField "Graphic I/O field_3" at 215,275 size 50x50; PictureList "Bombas"
      ProcessValue <- "UDT_Objetos_Bombas_BC-08_estado"
   GraphicIOField "Graphic I/O field_4" at 247,212 size 50x50; PictureList "Dosificadoras"
      ProcessValue <- "UDT_Objetos_Dosificadoras_BD-HIP-01_estado"
   GraphicIOField "Graphic I/O field_5" at 288,350 size 50x50; PictureList "Blower"
      ProcessValue <- "UDT_Objetos_Equipos_Especiales_BLW-01_estado"
   GraphicIOField "Graphic I/O field_6" at 406,311 size 30x30; PictureList "Valvulas"
      ProcessValue <- "UDT_Objetos_Valvulas_VM-31_estado"
   GraphicIOField "Graphic I/O field_7" at 403,342 size 30x30; PictureList "Valvulas"
      ProcessValue <- "UDT_Objetos_Valvulas_VM-32_estado"
   GraphicIOField "Graphic I/O field_8" at 471,394 size 30x30; PictureList "Valvulas"
      ProcessValue <- "UDT_Objetos_Valvulas_VM-41_estado"
   GraphicIOField "Graphic I/O field_9" at 586,353 size 30x30; PictureList "ValvulasRotadas"
      ProcessValue <- "UDT_Objetos_Valvulas_VM-40_estado"
   GraphicIOField "Graphic I/O field_10" at 693,205 size 30x30; PictureList "ValvulasRotadas"
      ProcessValue <- "UDT_Objetos_Valvulas_VM-34_estado"
   GraphicIOField "Graphic I/O field_11" at 637,310 size 30x30; PictureList "Valvulas"
      ProcessValue <- "UDT_Objetos_Valvulas_VM-33_estado"
   IOField "I/O field_6" at 276,298 size 71x19; FormatPattern 9999; Unit  m3/h
      ProcessValue <- "UDT_Objetos_Flujo_FI-06_flujo"
   IOField "I/O field_1" at 345,298 size 59x19; FormatPattern 9999; Unit  Bar
      ProcessValue <- "UDT_Objetos_Presion_PT-05_presion"
   Bar "Bar_1" at 134,209 size 14x93; MinimumValue 0; MaximumValue 100
      ProcessValue <- "UDT_Objetos_Nivel_RAD-04_nivel_porcentaje"
   Button "Button_4" at 718,155 size 72x39; TextOff 'OSMOSIS'
      on Click: ActivateScreen("2Osmosis", 0)
   Button "Button_5" at 713,395 size 72x39; TextOff 'ULTRA FILTRADA'
      on Click: ActivateScreen("1Ultrafiltrada", 0)
   IOField "I/O field_2" at 74,236 size 58x19; FormatPattern 9999; Unit  m3
      ProcessValue <- "UDT_Objetos_Nivel_RAD-04_nivel_volumen"
   IOField "I/O field_3" at 74,256 size 58x19; FormatPattern 999; Unit  m
      ProcessValue <- "UDT_Objetos_Nivel_RAD-04_nivel"

screen "Manual" 800x480, template "Alarmas"
   Button "Button_1" at 23,34 size 96x32; TextOff 'BC-08'
      ProcessValue <- "UDT_Objetos_Bombas_BC-11_frecuencia"
      on Click: InvertBit("UDT_Objetos_Bombas_BC-08_control")
      Appearance <- "UDT_Objetos_Bombas_BC-08_estado"
   Button "Button_2" at 23,83 size 96x32; TextOff 'BC-09'
      ProcessValue <- "UDT_Objetos_Bombas_BC-11_frecuencia"
      on Click: InvertBit("UDT_Objetos_Bombas_BC-09_control")
      Appearance <- "UDT_Objetos_Bombas_BC-09_estado"
   Button "Button_3" at 23,132 size 96x32; TextOff 'BC-10'
      ProcessValue <- "UDT_Objetos_Bombas_BC-11_frecuencia"
      on Click: InvertBit("UDT_Objetos_Bombas_BC-10_control")
      Appearance <- "UDT_Objetos_Bombas_BC-10_estado"
   Button "Button_4" at 23,181 size 96x32; TextOff 'BC-11'
      ProcessValue <- "UDT_Objetos_Bombas_BC-11_frecuencia"
      on Click: InvertBit("UDT_Objetos_Bombas_BC-11_control")
      Appearance <- "UDT_Objetos_Bombas_BC-11_estado"
   Button "Button_5" at 23,280 size 96x32; TextOff 'BC-12'
      ProcessValue <- "UDT_Objetos_Bombas_BC-11_frecuencia"
      on Click: InvertBit("UDT_Objetos_Bombas_BC-12_control")
      Appearance <- "UDT_Objetos_Bombas_BC-12_estado"
   Button "Button_6" at 23,329 size 96x32; TextOff 'BC-13'
      ProcessValue <- "UDT_Objetos_Bombas_BC-11_frecuencia"
      on Click: InvertBit("UDT_Objetos_Bombas_BC-13_control")
      Appearance <- "UDT_Objetos_Bombas_BC-13_estado"
   IOField "I/O field_1" at 23,215 size 96x32; FormatPattern 99
      ProcessValue <- "UDT_Objetos_Bombas_BC-11_frecuencia"
      Appearance <- "UDT_Objetos_Bombas_BC-11_estado"
   Button "Button_7" at 23,379 size 96x32; TextOff 'BC-14'
      ProcessValue <- "UDT_Objetos_Bombas_BC-11_frecuencia"
      on Click: InvertBit("UDT_Objetos_Bombas_BC-14_control")
      Appearance <- "UDT_Objetos_Bombas_BC-14_estado"
   Button "Button_8" at 154,34 size 96x32; TextOff 'BD-AI-01'
      ProcessValue <- "UDT_Objetos_Bombas_BC-11_frecuencia"
      on Click: InvertBit("UDT_Objetos_Dosificadoras_BD-AI-01_control")
      Appearance <- "UDT_Objetos_Dosificadoras_BD-AI-01_estado"
   Button "Button_9" at 154,83 size 96x32; TextOff 'BD-BIO-01'
      ProcessValue <- "UDT_Objetos_Bombas_BC-11_frecuencia"
      on Click: InvertBit("UDT_Objetos_Dosificadoras_BD-BIO-01_control")
      Appearance <- "UDT_Objetos_Dosificadoras_BD-BIO-01_estado"
   Button "Button_10" at 154,132 size 96x32; TextOff 'BD-HIP-01'
      ProcessValue <- "UDT_Objetos_Bombas_BC-11_frecuencia"
      on Click: InvertBit("UDT_Objetos_Dosificadoras_BD-HIP-01_control")
      Appearance <- "UDT_Objetos_Dosificadoras_BD-HIP-01_estado"
   Button "Button_11" at 154,181 size 96x32; TextOff 'BD-HIP-02'
      ProcessValue <- "UDT_Objetos_Bombas_BC-11_frecuencia"
      on Click: InvertBit("UDT_Objetos_Dosificadoras_BD-HIP-02_control")
      Appearance <- "UDT_Objetos_Dosificadoras_BD-HIP-02_estado"
   Button "Button_12" at 154,280 size 96x32; TextOff 'BD-UF-01'
      ProcessValue <- "UDT_Objetos_Bombas_BC-11_frecuencia"
      on Click: InvertBit("UDT_Objetos_Dosificadoras_BD-UF-01_control")
      Appearance <- "UDT_Objetos_Dosificadoras_BD-UF-01_estado"
   Button "Button_13" at 154,329 size 96x32; TextOff 'BLW-01'
      ProcessValue <- "UDT_Objetos_Bombas_BC-11_frecuencia"
      on Click: InvertBit("UDT_Objetos_Equipos_Especiales_BLW-01_control")
      Appearance <- "UDT_Objetos_Equipos_Especiales_BLW-01_estado"
   Button "Button_14" at 154,379 size 96x32; TextOff 'UV-01'
      ProcessValue <- "UDT_Objetos_Bombas_BC-11_frecuencia"
      on Click: InvertBit("UDT_Objetos_Equipos_Especiales_UV-01_control")
      Appearance <- "UDT_Objetos_Equipos_Especiales_UV-01_estado"
   Button "Button_15" at 154,230 size 96x32; TextOff 'BD-MBI-01'
      ProcessValue <- "UDT_Objetos_Bombas_BC-11_frecuencia"
      on Click: InvertBit("UDT_Objetos_Dosificadoras_BD-MBI-01_control")
      Appearance <- "UDT_Objetos_Dosificadoras_BD-MBI-01_estado"
   Button "Button_16" at 285,34 size 96x32; TextOff 'VM-27'
      ProcessValue <- "UDT_Objetos_Bombas_BC-11_frecuencia"
      on Click: InvertBit("UDT_Objetos_Valvulas_VM-27_control")
      Appearance <- "UDT_Objetos_Valvulas_VM-27_estado"
   Button "Button_17" at 285,83 size 96x32; TextOff 'VM-29'
      ProcessValue <- "UDT_Objetos_Bombas_BC-11_frecuencia"
      on Click: InvertBit("UDT_Objetos_Valvulas_VM-29_control")
      Appearance <- "UDT_Objetos_Valvulas_VM-29_estado"
   Button "Button_18" at 285,132 size 96x32; TextOff 'VM-31'
      ProcessValue <- "UDT_Objetos_Bombas_BC-11_frecuencia"
      on Click: InvertBit("UDT_Objetos_Valvulas_VM-31_control")
      Appearance <- "UDT_Objetos_Valvulas_VM-31_estado"
   Button "Button_19" at 285,181 size 96x32; TextOff 'VM-32'
      ProcessValue <- "UDT_Objetos_Bombas_BC-11_frecuencia"
      on Click: InvertBit("UDT_Objetos_Valvulas_VM-32_control")
      Appearance <- "UDT_Objetos_Valvulas_VM-32_estado"
   Button "Button_20" at 285,280 size 96x32; TextOff 'VM-34'
      ProcessValue <- "UDT_Objetos_Bombas_BC-11_frecuencia"
      on Click: InvertBit("UDT_Objetos_Valvulas_VM-34_control")
      Appearance <- "UDT_Objetos_Valvulas_VM-34_estado"
   Button "Button_21" at 285,329 size 96x32; TextOff 'VM-35'
      ProcessValue <- "UDT_Objetos_Bombas_BC-11_frecuencia"
      on Click: InvertBit("UDT_Objetos_Valvulas_VM-35_control")
      Appearance <- "UDT_Objetos_Valvulas_VM-35_estado"
   Button "Button_22" at 285,230 size 96x32; TextOff 'VM-33'
      ProcessValue <- "UDT_Objetos_Bombas_BC-11_frecuencia"
      on Click: InvertBit("UDT_Objetos_Valvulas_VM-33_control")
      Appearance <- "UDT_Objetos_Valvulas_VM-33_estado"
   Button "Button_23" at 285,379 size 96x32; TextOff 'VM-36'
      ProcessValue <- "UDT_Objetos_Bombas_BC-11_frecuencia"
      on Click: InvertBit("UDT_Objetos_Valvulas_VM-36_control")
      Appearance <- "UDT_Objetos_Valvulas_VM-36_estado"
   Button "Button_24" at 417,34 size 96x32; TextOff 'VM-39'
      ProcessValue <- "UDT_Objetos_Bombas_BC-11_frecuencia"
      on Click: InvertBit("UDT_Objetos_Valvulas_VM-39_control")
      Appearance <- "UDT_Objetos_Valvulas_VM-39_estado"
   Button "Button_25" at 417,83 size 96x32; TextOff 'VM-40'
      ProcessValue <- "UDT_Objetos_Bombas_BC-11_frecuencia"
      on Click: InvertBit("UDT_Objetos_Valvulas_VM-40_control")
      Appearance <- "UDT_Objetos_Valvulas_VM-40_estado"
   Button "Button_26" at 417,132 size 96x32; TextOff 'VM-41'
      ProcessValue <- "UDT_Objetos_Bombas_BC-11_frecuencia"
      on Click: InvertBit("UDT_Objetos_Valvulas_VM-41_control")
      Appearance <- "UDT_Objetos_Valvulas_VM-41_estado"
   Button "Button_27" at 417,181 size 96x32; TextOff 'VM-42'
      ProcessValue <- "UDT_Objetos_Bombas_BC-11_frecuencia"
      on Click: InvertBit("UDT_Objetos_Valvulas_VM-42_control")
      Appearance <- "UDT_Objetos_Valvulas_VM-42_estado"
   Button "Button_28" at 417,280 size 96x32; TextOff 'VM-46'
      ProcessValue <- "UDT_Objetos_Bombas_BC-11_frecuencia"
      on Click: InvertBit("UDT_Objetos_Valvulas_VM-46_control")
      Appearance <- "UDT_Objetos_Valvulas_VM-46_estado"
   Button "Button_29" at 417,329 size 96x32; TextOff 'VM-47'
      ProcessValue <- "UDT_Objetos_Bombas_BC-11_frecuencia"
      on Click: InvertBit("UDT_Objetos_Valvulas_VM-47_control")
      Appearance <- "UDT_Objetos_Valvulas_VM-47_estado"
   Button "Button_30" at 417,230 size 96x32; TextOff 'VM-45'
      ProcessValue <- "UDT_Objetos_Bombas_BC-11_frecuencia"
      on Click: InvertBit("UDT_Objetos_Valvulas_VM-45_control")
      Appearance <- "UDT_Objetos_Valvulas_VM-45_estado"
   Button "Button_31" at 417,379 size 96x32; TextOff 'VM-48'
      ProcessValue <- "UDT_Objetos_Bombas_BC-11_frecuencia"
      on Click: InvertBit("UDT_Objetos_Valvulas_VM-48_control")
      Appearance <- "UDT_Objetos_Valvulas_VM-48_estado"
   Button "Button_32" at 548,34 size 96x32; TextOff 'VM-49'
      ProcessValue <- "UDT_Objetos_Bombas_BC-11_frecuencia"
      on Click: InvertBit("UDT_Objetos_Valvulas_VM-49_control")
      Appearance <- "UDT_Objetos_Valvulas_VM-49_estado"
   Button "Button_33" at 548,83 size 96x32; TextOff 'VM-50'
      ProcessValue <- "UDT_Objetos_Bombas_BC-11_frecuencia"
      on Click: InvertBit("UDT_Objetos_Valvulas_VM-50_control")
      Appearance <- "UDT_Objetos_Valvulas_VM-50_estado"
   Button "Button_34" at 548,132 size 96x32; TextOff 'VM-51'
      ProcessValue <- "UDT_Objetos_Bombas_BC-11_frecuencia"
      on Click: InvertBit("UDT_Objetos_Valvulas_VM-51_control")
      Appearance <- "UDT_Objetos_Valvulas_VM-51_estado"
   Button "Button_35" at 548,181 size 96x32; TextOff 'VM-52'
      ProcessValue <- "UDT_Objetos_Bombas_BC-11_frecuencia"
      on Click: InvertBit("UDT_Objetos_Valvulas_VM-52_control")
      Appearance <- "UDT_Objetos_Valvulas_VM-52_estado"
   Button "Button_36" at 548,280 size 96x32; TextOff 'VM-56'
      ProcessValue <- "UDT_Objetos_Bombas_BC-11_frecuencia"
      on Click: InvertBit("UDT_Objetos_Valvulas_VM-56_control")
      Appearance <- "UDT_Objetos_Valvulas_VM-56_estado"
   Button "Button_37" at 548,329 size 96x32; TextOff 'VM-57'
      ProcessValue <- "UDT_Objetos_Bombas_BC-11_frecuencia"
      on Click: InvertBit("UDT_Objetos_Valvulas_VM-57_control")
      Appearance <- "UDT_Objetos_Valvulas_VM-57_estado"
   Button "Button_38" at 548,230 size 96x32; TextOff 'VM-53'
      ProcessValue <- "UDT_Objetos_Bombas_BC-11_frecuencia"
      on Click: InvertBit("UDT_Objetos_Valvulas_VM-53_control")
      Appearance <- "UDT_Objetos_Valvulas_VM-53_estado"
   Button "Button_39" at 548,379 size 96x32; TextOff 'VM-58'
      ProcessValue <- "UDT_Objetos_Bombas_BC-11_frecuencia"
      on Click: InvertBit("UDT_Objetos_Valvulas_VM-58_control")
      Appearance <- "UDT_Objetos_Valvulas_VM-58_estado"
   Button "Button_40" at 680,34 size 96x32; TextOff 'VM-61'
      ProcessValue <- "UDT_Objetos_Bombas_BC-11_frecuencia"
      on Click: InvertBit("UDT_Objetos_Valvulas_VM-61_control")
      Appearance <- "UDT_Objetos_Valvulas_VM-61_estado"
   Button "Button_41" at 680,83 size 96x32; TextOff 'VM-62'
      ProcessValue <- "UDT_Objetos_Bombas_BC-11_frecuencia"
      on Click: InvertBit("UDT_Objetos_Valvulas_VM-62_control")
      Appearance <- "UDT_Objetos_Valvulas_VM-62_estado"
   Button "Button_42" at 680,132 size 96x32; TextOff 'VM-63'
      ProcessValue <- "UDT_Objetos_Bombas_BC-11_frecuencia"
      on Click: InvertBit("UDT_Objetos_Valvulas_VM-63_control")
      Appearance <- "UDT_Objetos_Valvulas_VM-63_estado"

screen "BASE" 800x480, template "Template_1"
   Button "Button_1" at 23,34 size 96x32; TextOff 'BC-08'
      on Click: InvertBit("UDT_Objetos_Bombas_BC-08_control")
      ProcessValue <- "UDT_Objetos_Bombas_BC-11_frecuencia"
      Appearance <- "UDT_Objetos_Bombas_BC-08_estado"
   Button "Button_2" at 23,83 size 96x32; TextOff 'BC-09'
      on Click: InvertBit("UDT_Objetos_Bombas_BC-09_control")
      ProcessValue <- "UDT_Objetos_Bombas_BC-11_frecuencia"
      Appearance <- "UDT_Objetos_Bombas_BC-09_estado"
   Button "Button_3" at 23,132 size 96x32; TextOff 'BC-10'
      on Click: InvertBit("UDT_Objetos_Bombas_BC-10_control")
      ProcessValue <- "UDT_Objetos_Bombas_BC-11_frecuencia"
      Appearance <- "UDT_Objetos_Bombas_BC-10_estado"
   Button "Button_4" at 23,181 size 96x32; TextOff 'BC-11'
      on Click: InvertBit("UDT_Objetos_Bombas_BC-11_control")
      ProcessValue <- "UDT_Objetos_Bombas_BC-11_frecuencia"
      Appearance <- "UDT_Objetos_Bombas_BC-11_estado"
   Button "Button_5" at 23,280 size 96x32; TextOff 'BC-12'
      on Click: InvertBit("UDT_Objetos_Bombas_BC-12_control")
      ProcessValue <- "UDT_Objetos_Bombas_BC-11_frecuencia"
      Appearance <- "UDT_Objetos_Bombas_BC-12_estado"
   Button "Button_6" at 23,329 size 96x32; TextOff 'BC-13'
      on Click: InvertBit("UDT_Objetos_Bombas_BC-13_control")
      ProcessValue <- "UDT_Objetos_Bombas_BC-11_frecuencia"
      Appearance <- "UDT_Objetos_Bombas_BC-13_estado"
   IOField "I/O field_1" at 23,215 size 96x32; FormatPattern 99
      ProcessValue <- "UDT_Objetos_Bombas_BC-11_frecuencia"
      Appearance <- "UDT_Objetos_Valvulas_VM-33_estado"
   Button "Button_7" at 23,379 size 96x32; TextOff 'BC-14'
      on Click: InvertBit("UDT_Objetos_Bombas_BC-14_control")
      ProcessValue <- "UDT_Objetos_Bombas_BC-11_frecuencia"
      Appearance <- "UDT_Objetos_Bombas_BC-14_estado"
   Button "Button_8" at 154,34 size 96x32; TextOff 'BD-AI-01'
      on Click: InvertBit("UDT_Objetos_Dosificadoras_BD-AI-01_control")
      ProcessValue <- "UDT_Objetos_Bombas_BC-11_frecuencia"
      Appearance <- "UDT_Objetos_Dosificadoras_BD-AI-01_estado"
   Button "Button_9" at 154,83 size 96x32; TextOff 'BD-BIO-01'
      on Click: InvertBit("UDT_Objetos_Dosificadoras_BD-BIO-01_control")
      ProcessValue <- "UDT_Objetos_Bombas_BC-11_frecuencia"
      Appearance <- "UDT_Objetos_Dosificadoras_BD-BIO-01_estado"
   Button "Button_10" at 154,132 size 96x32; TextOff 'BD-HIP-01'
      on Click: InvertBit("UDT_Objetos_Dosificadoras_BD-HIP-01_control")
      ProcessValue <- "UDT_Objetos_Bombas_BC-11_frecuencia"
      Appearance <- "UDT_Objetos_Dosificadoras_BD-HIP-01_estado"
   Button "Button_11" at 154,181 size 96x32; TextOff 'BD-HIP-02'
      on Click: InvertBit("UDT_Objetos_Dosificadoras_BD-HIP-02_control")
      ProcessValue <- "UDT_Objetos_Bombas_BC-11_frecuencia"
      Appearance <- "UDT_Objetos_Dosificadoras_BD-HIP-02_estado"
   Button "Button_12" at 154,280 size 96x32; TextOff 'BD-UF-01'
      on Click: InvertBit("UDT_Objetos_Dosificadoras_BD-UF-01_control")
      ProcessValue <- "UDT_Objetos_Bombas_BC-11_frecuencia"
      Appearance <- "UDT_Objetos_Dosificadoras_BD-UF-01_estado"
   Button "Button_13" at 154,329 size 96x32; TextOff 'BLW-01'
      on Click: InvertBit("UDT_Objetos_Equipos_Especiales_BLW-01_control")
      ProcessValue <- "UDT_Objetos_Bombas_BC-11_frecuencia"
      Appearance <- "UDT_Objetos_Equipos_Especiales_BLW-01_estado"
   Button "Button_14" at 154,379 size 96x32; TextOff 'UV-01'
      on Click: InvertBit("UDT_Objetos_Equipos_Especiales_UV-01_control")
      ProcessValue <- "UDT_Objetos_Bombas_BC-11_frecuencia"
      Appearance <- "UDT_Objetos_Equipos_Especiales_UV-01_estado"
   Button "Button_15" at 154,230 size 96x32; TextOff 'BD-MBI-01'
      on Click: InvertBit("UDT_Objetos_Dosificadoras_BD-MBI-01_control")
      ProcessValue <- "UDT_Objetos_Bombas_BC-11_frecuencia"
      Appearance <- "UDT_Objetos_Dosificadoras_BD-MBI-01_estado"
   Button "Button_16" at 285,34 size 96x32; TextOff 'VM-27'
      on Click: InvertBit("UDT_Objetos_Valvulas_VM-27_control")
      ProcessValue <- "UDT_Objetos_Bombas_BC-11_frecuencia"
      Appearance <- "UDT_Objetos_Valvulas_VM-27_estado"
   Button "Button_17" at 285,83 size 96x32; TextOff 'VM-29'
      on Click: InvertBit("UDT_Objetos_Valvulas_VM-29_control")
      ProcessValue <- "UDT_Objetos_Bombas_BC-11_frecuencia"
      Appearance <- "UDT_Objetos_Valvulas_VM-29_estado"
   Button "Button_18" at 285,132 size 96x32; TextOff 'VM-31'
      on Click: InvertBit("UDT_Objetos_Valvulas_VM-31_control")
      ProcessValue <- "UDT_Objetos_Bombas_BC-11_frecuencia"
      Appearance <- "UDT_Objetos_Valvulas_VM-31_estado"
   Button "Button_19" at 285,181 size 96x32; TextOff 'VM-32'
      on Click: InvertBit("UDT_Objetos_Valvulas_VM-32_control")
      ProcessValue <- "UDT_Objetos_Bombas_BC-11_frecuencia"
      Appearance <- "UDT_Objetos_Valvulas_VM-32_estado"
   Button "Button_20" at 285,280 size 96x32; TextOff 'VM-34'
      on Click: InvertBit("UDT_Objetos_Valvulas_VM-34_control")
      ProcessValue <- "UDT_Objetos_Bombas_BC-11_frecuencia"
      Appearance <- "UDT_Objetos_Valvulas_VM-34_estado"
   Button "Button_21" at 285,329 size 96x32; TextOff 'VM-35'
      on Click: InvertBit("UDT_Objetos_Valvulas_VM-35_control")
      ProcessValue <- "UDT_Objetos_Bombas_BC-11_frecuencia"
      Appearance <- "UDT_Objetos_Valvulas_VM-35_estado"
   Button "Button_22" at 285,230 size 96x32; TextOff 'VM-33'
      on Click: InvertBit("UDT_Objetos_Valvulas_VM-33_control")
      ProcessValue <- "UDT_Objetos_Bombas_BC-11_frecuencia"
      Appearance <- "UDT_Objetos_Valvulas_VM-33_estado"
   Button "Button_23" at 285,379 size 96x32; TextOff 'VM-36'
      on Click: InvertBit("UDT_Objetos_Valvulas_VM-36_control")
      ProcessValue <- "UDT_Objetos_Bombas_BC-11_frecuencia"
      Appearance <- "UDT_Objetos_Valvulas_VM-36_estado"
   Button "Button_24" at 417,34 size 96x32; TextOff 'VM-39'
      on Click: InvertBit("UDT_Objetos_Valvulas_VM-39_control")
      ProcessValue <- "UDT_Objetos_Bombas_BC-11_frecuencia"
      Appearance <- "UDT_Objetos_Valvulas_VM-39_estado"
   Button "Button_25" at 417,83 size 96x32; TextOff 'VM-40'
      on Click: InvertBit("UDT_Objetos_Valvulas_VM-40_control")
      ProcessValue <- "UDT_Objetos_Bombas_BC-11_frecuencia"
      Appearance <- "UDT_Objetos_Valvulas_VM-40_estado"
   Button "Button_26" at 417,132 size 96x32; TextOff 'VM-41'
      on Click: InvertBit("UDT_Objetos_Valvulas_VM-41_control")
      ProcessValue <- "UDT_Objetos_Bombas_BC-11_frecuencia"
      Appearance <- "UDT_Objetos_Valvulas_VM-41_estado"
   Button "Button_27" at 417,181 size 96x32; TextOff 'VM-42'
      on Click: InvertBit("UDT_Objetos_Valvulas_VM-42_control")
      ProcessValue <- "UDT_Objetos_Bombas_BC-11_frecuencia"
      Appearance <- "UDT_Objetos_Valvulas_VM-42_estado"
   Button "Button_28" at 417,280 size 96x32; TextOff 'VM-46'
      on Click: InvertBit("UDT_Objetos_Valvulas_VM-46_control")
      ProcessValue <- "UDT_Objetos_Bombas_BC-11_frecuencia"
      Appearance <- "UDT_Objetos_Valvulas_VM-46_estado"
   Button "Button_29" at 417,329 size 96x32; TextOff 'VM-47'
      on Click: InvertBit("UDT_Objetos_Valvulas_VM-47_control")
      ProcessValue <- "UDT_Objetos_Bombas_BC-11_frecuencia"
      Appearance <- "UDT_Objetos_Valvulas_VM-47_estado"
   Button "Button_30" at 417,230 size 96x32; TextOff 'VM-45'
      on Click: InvertBit("UDT_Objetos_Valvulas_VM-45_control")
      ProcessValue <- "UDT_Objetos_Bombas_BC-11_frecuencia"
      Appearance <- "UDT_Objetos_Valvulas_VM-45_estado"
   Button "Button_31" at 417,379 size 96x32; TextOff 'VM-48'
      on Click: InvertBit("UDT_Objetos_Valvulas_VM-48_control")
      ProcessValue <- "UDT_Objetos_Bombas_BC-11_frecuencia"
      Appearance <- "UDT_Objetos_Valvulas_VM-48_estado"
   Button "Button_32" at 548,34 size 96x32; TextOff 'VM-49'
      on Click: InvertBit("UDT_Objetos_Valvulas_VM-49_control")
      ProcessValue <- "UDT_Objetos_Bombas_BC-11_frecuencia"
      Appearance <- "UDT_Objetos_Valvulas_VM-49_estado"
   Button "Button_33" at 548,83 size 96x32; TextOff 'VM-50'
      on Click: InvertBit("UDT_Objetos_Valvulas_VM-50_control")
      ProcessValue <- "UDT_Objetos_Bombas_BC-11_frecuencia"
      Appearance <- "UDT_Objetos_Valvulas_VM-50_estado"
   Button "Button_34" at 548,132 size 96x32; TextOff 'VM-51'
      on Click: InvertBit("UDT_Objetos_Valvulas_VM-51_control")
      ProcessValue <- "UDT_Objetos_Bombas_BC-11_frecuencia"
      Appearance <- "UDT_Objetos_Valvulas_VM-51_estado"
   Button "Button_35" at 548,181 size 96x32; TextOff 'VM-52'
      on Click: InvertBit("UDT_Objetos_Valvulas_VM-52_control")
      ProcessValue <- "UDT_Objetos_Bombas_BC-11_frecuencia"
      Appearance <- "UDT_Objetos_Valvulas_VM-52_estado"
   Button "Button_36" at 548,280 size 96x32; TextOff 'VM-56'
      on Click: InvertBit("UDT_Objetos_Valvulas_VM-56_control")
      ProcessValue <- "UDT_Objetos_Bombas_BC-11_frecuencia"
      Appearance <- "UDT_Objetos_Valvulas_VM-56_estado"
   Button "Button_37" at 548,329 size 96x32; TextOff 'VM-57'
      on Click: InvertBit("UDT_Objetos_Valvulas_VM-57_control")
      ProcessValue <- "UDT_Objetos_Bombas_BC-11_frecuencia"
      Appearance <- "UDT_Objetos_Valvulas_VM-57_estado"
   Button "Button_38" at 548,230 size 96x32; TextOff 'VM-53'
      on Click: InvertBit("UDT_Objetos_Valvulas_VM-53_control")
      ProcessValue <- "UDT_Objetos_Bombas_BC-11_frecuencia"
      Appearance <- "UDT_Objetos_Valvulas_VM-53_estado"
   Button "Button_39" at 548,379 size 96x32; TextOff 'VM-58'
      on Click: InvertBit("UDT_Objetos_Valvulas_VM-58_control")
      ProcessValue <- "UDT_Objetos_Bombas_BC-11_frecuencia"
      Appearance <- "UDT_Objetos_Valvulas_VM-58_estado"
   Button "Button_40" at 680,34 size 96x32; TextOff 'VM-61'
      on Click: InvertBit("UDT_Objetos_Valvulas_VM-61_control")
      ProcessValue <- "UDT_Objetos_Bombas_BC-11_frecuencia"
      Appearance <- "UDT_Objetos_Valvulas_VM-61_estado"
   Button "Button_41" at 680,83 size 96x32; TextOff 'VM-62'
      on Click: InvertBit("UDT_Objetos_Valvulas_VM-62_control")
      ProcessValue <- "UDT_Objetos_Bombas_BC-11_frecuencia"
      Appearance <- "UDT_Objetos_Valvulas_VM-62_estado"
   Button "Button_42" at 680,132 size 50x50; TextOff 'VM-63'
      on Click: InvertBit("UDT_Objetos_Valvulas_VM-63_control")
      ProcessValue <- "UDT_Objetos_Bombas_BC-11_frecuencia"
      Appearance <- "UDT_Objetos_Valvulas_VM-63_estado"

screen "1Ultrafiltrada" 800x480, template "Template_1"
   Button "Button_1" at 694,0 size 106x56; TextOff 'AJUSTES'
      on Click: ActivateScreen("Configuraciones", 0)
   AlarmView "Alarm view_1" at 111,0 size 584x56
   GraphicView "Graphic view_1" at 0,0 size 112x56; Picture "Coca-Cola_Femsa_Logo"
   GraphicView "Graphic view_2" at 0,107 size 800x332; Picture "ULTRAFILTRADA_1"
   GraphicIOField "Graphic I/O field_6" at 147,268 size 30x30; PictureList "Valvulas"
      ProcessValue <- "UDT_Objetos_Valvulas_VM-35_estado"
   GraphicIOField "Graphic I/O field_1" at 83,301 size 30x30; PictureList "ValvulasRotadas"
      ProcessValue <- "UDT_Objetos_Valvulas_VM-39_estado"
   GraphicIOField "Graphic I/O field_2" at 203,229 size 30x30; PictureList "Valvulas"
      ProcessValue <- "UDT_Objetos_Valvulas_VM-36_estado"
   GraphicIOField "Graphic I/O field_3" at 219,376 size 30x30; PictureList "Valvulas"
      ProcessValue <- "UDT_Objetos_Valvulas_VM-42_estado"
   GraphicIOField "Graphic I/O field_4" at 277,357 size 50x50; PictureList "BombaDerechas"
      ProcessValue <- "UDT_Objetos_Bombas_BC-09_estado"
   GraphicIOField "Graphic I/O field_5" at 469,357 size 50x50; PictureList "BombasIzquierdas"
      ProcessValue <- "UDT_Objetos_Bombas_BC-10_estado"
   GraphicIOField "Graphic I/O field_7" at 650,247 size 30x30; PictureList "Valvulas"
      ProcessValue <- "UDT_Objetos_Valvulas_VM-48_estado"
   GraphicIOField "Graphic I/O field_8" at 521,136 size 50x50; PictureList "DosificadorasIzquierdas"
      ProcessValue <- "UDT_Objetos_Dosificadoras_BD-MBI-01_estado"
   GraphicIOField "Graphic I/O field_9" at 621,358 size 30x30; PictureList "ValvulasRotadas"
      ProcessValue <- "UDT_Objetos_Valvulas_VM-46_estado"
   IOField "I/O field_6" at 254,161 size 71x19; FormatPattern 9999; Unit  m3/h
      ProcessValue <- "UDT_Objetos_Flujo_FI-07_flujo"
   IOField "I/O field_1" at 108,218 size 59x19; FormatPattern 9999; Unit  Bar
      ProcessValue <- "UDT_Objetos_Presion_PT-06_presion"
   Button "Button_4" at 9,203 size 85x39; TextOff 'ULTRA FILTRACION'
      on Click: ActivateScreen("0Ultrafiltracion", 0)
   Button "Button_3" at 9,356 size 85x39; TextOff 'ULTRA FILTRACION'
      on Click: ActivateScreen("0Ultrafiltracion", 0)
   Button "Button_5" at 694,281 size 85x39; TextOff 'OSMOSIS'
      on Click: ActivateScreen("2Osmosis", 0)
   IOField "I/O field_2" at 495,294 size 71x19; FormatPattern 9999; Unit  m3/h
      ProcessValue <- "UDT_Objetos_Flujo_FI-08_flujo"
   IOField "I/O field_3" at 576,294 size 65x19; FormatPattern s9999; Unit  mV
      ProcessValue <- "UDT_Objetos_Sensores_Especiales_ORP-01_medicion"
   Bar "Bar_1" at 431,273 size 14x133; MinimumValue 0; MaximumValue 100
      ProcessValue <- "UDT_Objetos_Nivel_PT-07_nivel_porcentaje"
   IOField "I/O field_4" at 358,320 size 58x19; FormatPattern 9999; Unit  m3
      ProcessValue <- "UDT_Objetos_Nivel_PT-07_nivel_volumen"
   IOField "I/O field_5" at 358,340 size 58x19; FormatPattern 999; Unit  m
      ProcessValue <- "UDT_Objetos_Nivel_PT-07_nivel"

screen "2Osmosis" 800x480, template "Template_1"
   Button "Button_1" at 694,0 size 106x56; TextOff 'AJUSTES'
      on Click: ActivateScreen("Configuraciones", 0)
   AlarmView "Alarm view_1" at 111,0 size 584x56
   GraphicView "Graphic view_1" at 0,0 size 112x56; Picture "Coca-Cola_Femsa_Logo"
   GraphicView "Graphic view_2" at 0,107 size 800x332; Picture "OSMOSIS_2"
   Button "Button_4" at 222,336 size 50x50; TextOff 'Text'; PictureList "DosificadorasDerecha"
      ProcessValue <- "UDT_Objetos_Dosificadoras_BD-AI-01_estado"
   Button "Button_7" at 488,307 size 30x30; TextOff 'Text'; PictureList "Valvulas"
      ProcessValue <- "UDT_Objetos_Valvulas_VM-47_estado"
   Button "Button_11" at 521,349 size 30x30; TextOff 'Text'; PictureList "ValvulasRotadas"
      ProcessValue <- "UDT_Objetos_Valvulas_VM-56_estado"
   GraphicIOField "Graphic I/O field_2" at 333,251 size 90x90; PictureList "BombaGrande"
      ProcessValue <- "UDT_Objetos_Bombas_BC-11_estado"
   GraphicIOField "Graphic I/O field_1" at 222,336 size 50x50; PictureList "DosificadorasDerecha"
      ProcessValue <- "UDT_Objetos_Valvulas_VM-36_estado"
   GraphicIOField "Graphic I/O field_3" at 231,254 size 30x30; PictureList "ValvulasRotadas"
      ProcessValue <- "UDT_Objetos_Valvulas_VM-45_estado"
   GraphicIOField "Graphic I/O field_5" at 521,349 size 30x30; PictureList "ValvulasRotadas"
      ProcessValue <- "UDT_Objetos_Valvulas_VM-56_estado"
   IOField "I/O field_1" at 299,296 size 59x19; FormatPattern 9999; Unit  Bar
      ProcessValue <- "UDT_Objetos_Presion_PT-08_presion"
   IOField "I/O field_2" at 403,295 size 59x19; FormatPattern 9999; Unit  Bar
      ProcessValue <- "UDT_Objetos_Presion_PT-09_presion"
   IOField "I/O field_3" at 672,287 size 59x19; FormatPattern 9999; Unit  Bar
      ProcessValue <- "UDT_Objetos_Presion_PT-10_presion"
   Button "Button_3" at 113,177 size 85x39; TextOff 'ULTRA FILTRACION'
      on Click: ActivateScreen("0Ultrafiltracion", 0)
   Button "Button_5" at 418,393 size 85x39; TextOff 'PERMEADO'
      on Click: ActivateScreen("4Permeado", 0)
   Button "Button_6" at 683,393 size 85x39; TextOff 'CAPTACION'
      on Click: ActivateScreen("5CaptacionRechazo", 0)
   Button "Button_8" at 518,393 size 85x39; TextOff 'CIP'
      on Click: ActivateScreen("3CIP UF", 0)
   Button "Button_12" at 114,237 size 85x39; TextOff 'ULTRA FILTRADA'
      on Click: ActivateScreen("1Ultrafiltrada", 0)
   IOField "I/O field_4" at 351,221 size 54x19; FormatPattern 9999; Unit  Hz
      ProcessValue <- "UDT_Objetos_Bombas_BC-11_frecuencia"

screen "3CIP UF" 800x480, template "Template_1"
   on GenerateScreen: SetTag("PantallaActual", 3)
   GraphicView "Graphic view_2" at 0,107 size 800x332; Picture "CIPUF_2"
   Button "Button_1" at 694,0 size 106x56; TextOff 'AJUSTES'
   AlarmView "Alarm view_1" at 111,0 size 584x56
   GraphicView "Graphic view_1" at 0,0 size 112x56; Picture "Coca-Cola_Femsa_Logo"
   Button "Button_2" at 694,56 size 106x56; TextOff 'MANUAL'
      on Click: ActivateScreen("Manual", 0)
   GraphicIOField "Graphic I/O field_4" at 341,342 size 50x50; PictureList "BombaDerechas"
      ProcessValue <- "UDT_Objetos_Bombas_BC-10_estado"
   GraphicIOField "Graphic I/O field_10" at 498,196 size 30x30; PictureList "ValvulasRotadas"
      ProcessValue <- "UDT_Objetos_Valvulas_VM-49_estado"
   GraphicIOField "Graphic I/O field_11" at 659,201 size 30x30; PictureList "Valvulas"
      ProcessValue <- "UDT_Objetos_Valvulas_VM-51_estado"
   GraphicIOField "Graphic I/O field_12" at 609,368 size 30x30; PictureList "ValvulasRotadas"
      ProcessValue <- "UDT_Objetos_Valvulas_VM-52_estado"
   GraphicIOField "Graphic I/O field_13" at 614,144 size 30x30; PictureList "Valvulas"
      ProcessValue <- "UDT_Objetos_Valvulas_VM-50_estado"
   Button "Button_5" at 399,132 size 85x39; TextOff 'OSMOSIS'
      on Click: ActivateScreen("2Osmosis", 0)
   Button "Button_3" at 714,171 size 85x39; TextOff 'CAPTACION'
      on Click: ActivateScreen("5CaptacionRechazo", 0)

screen "4Permeado" 800x480, template "Template_1"
   on GenerateScreen: SetTag("PantallaActual", 4)
   Button "Button_1" at 694,0 size 106x56; TextOff 'AJUSTES'
      on Click: ActivateScreen("Configuraciones", 0)
   AlarmView "Alarm view_1" at 111,0 size 584x56
   GraphicView "Graphic view_1" at 0,0 size 112x56; Picture "Coca-Cola_Femsa_Logo"
   GraphicView "Graphic view_2" at 0,107 size 800x332; Picture "PERMEADO_3"
   GraphicIOField "Graphic I/O field_3" at 276,210 size 30x30; PictureList "Valvulas"
      ProcessValue <- "UDT_Objetos_Valvulas_VM-63_estado"
   GraphicIOField "Graphic I/O field_1" at 238,146 size 30x30; PictureList "ValvulasRotadas"
      ProcessValue <- "UDT_Objetos_Valvulas_VM-57_estado"
   GraphicIOField "Graphic I/O field_2" at 22,384 size 30x30; PictureList "Valvulas"
      ProcessValue <- "UDT_Objetos_Valvulas_VM-58_estado"
   GraphicIOField "Graphic I/O field_4" at 185,372 size 50x50; PictureList "BombasIzquierdas"
      ProcessValue <- "UDT_Objetos_Bombas_BC-13_estado"
   GraphicIOField "Graphic I/O field_5" at 350,392 size 50x50; PictureList "DosificadorasDerecha"
      ProcessValue <- "UDT_Objetos_Dosificadoras_BD-HIP-02_estado"
   GraphicIOField "Graphic I/O field_6" at 431,300 size 30x30; PictureList "Valvulas"
      ProcessValue <- "UDT_Objetos_Valvulas_VM-61_estado"
   GraphicIOField "Graphic I/O field_7" at 492,259 size 30x30; PictureList "Valvulas"
      ProcessValue <- "UDT_Objetos_Valvulas_VM-62_estado"
   GraphicIOField "Graphic I/O field_8" at 600,231 size 50x50; PictureList "DosificadorasIzquierdas"
      ProcessValue <- "UDT_Objetos_Dosificadoras_BD-BIO-01_estado"
   GraphicIOField "Graphic I/O field_9" at 245,239 size 100x100; PictureList "Ultravioleta"
      ProcessValue <- "UDT_Objetos_Equipos_Especiales_UV-01_estado"
   IOField "I/O field_6" at 244,327 size 71x19; FormatPattern 9999; Unit  m3/h
      ProcessValue <- "UDT_Objetos_Flujo_FI-11_flujo"
   IOField "I/O field_2" at 252,308 size 63x19; FormatPattern 999; Unit  mg/L
      ProcessValue <- "UDT_Objetos_Sensores_Especiales_COT-01_medicion"
   IOField "I/O field_1" at 147,191 size 71x19; FormatPattern 9999; Unit  m3/h
      ProcessValue <- "UDT_Objetos_Flujo_FI-09_flujo"
   Button "Button_3" at 282,117 size 85x39; TextOff 'OSMOSIS'
      on Click: ActivateScreen("2Osmosis", 0)
   Button "Button_2" at 153,117 size 85x39; TextOff 'CIP'
      on Click: ActivateScreen("2Osmosis", 0)
   Bar "Bar_1" at 150,278 size 14x133; MinimumValue 0; MaximumValue 100
      ProcessValue <- "UDT_Objetos_Nivel_PT-12_nivel_porcentaje"
   IOField "I/O field_3" at 80,326 size 58x19; FormatPattern 9999; Unit  m3
      ProcessValue <- "UDT_Objetos_Nivel_PT-12_nivel_volumen"
   IOField "I/O field_4" at 94,346 size 44x19; FormatPattern 999; Unit  m
      ProcessValue <- "UDT_Objetos_Nivel_PT-12_nivel"
   Bar "Bar_2" at 776,311 size 14x90; MinimumValue 0; MaximumValue 100
      ProcessValue <- "UDT_Objetos_Nivel_RAD-05_nivel_porcentaje"
   IOField "I/O field_5" at 708,334 size 58x19; FormatPattern 9999; Unit  m3
      ProcessValue <- "UDT_Objetos_Nivel_RAD-05_nivel_volumen"
   IOField "I/O field_7" at 722,354 size 44x19; FormatPattern 999; Unit  m
      ProcessValue <- "UDT_Objetos_Nivel_RAD-05_nivel"
   Bar "Bar_3" at 628,312 size 14x90; MinimumValue 0; MaximumValue 100
      ProcessValue <- "UDT_Objetos_Nivel_RAD-06_nivel_porcentaje"
   IOField "I/O field_8" at 559,339 size 58x19; FormatPattern 9999; Unit  m3
      ProcessValue <- "UDT_Objetos_Nivel_RAD-06_nivel_volumen"
   IOField "I/O field_9" at 573,359 size 44x19; FormatPattern 999; Unit  m
      ProcessValue <- "UDT_Objetos_Nivel_RAD-06_nivel"

screen "5CaptacionRechazo" 800x480, template "Template_1"
   on GenerateScreen: SetTag("PantallaActual", 5)
   Button "Button_1" at 694,0 size 106x56; TextOff 'AJUSTES'
      on Click: ActivateScreen("Configuraciones", 0)
   AlarmView "Alarm view_1" at 111,0 size 584x56
   GraphicView "Graphic view_1" at 0,0 size 112x56; Picture "Coca-Cola_Femsa_Logo"
   GraphicView "Graphic view_2" at 0,107 size 800x332; Picture "CaptacionRechazo_1"
   GraphicIOField "Graphic I/O field_4" at 665,362 size 50x50; PictureList "BombasIzquierdas"
      ProcessValue <- "UDT_Objetos_Bombas_BC-14_estado"
   GraphicIOField "Graphic I/O field_7" at 379,278 size 30x30; PictureList "Valvulas"
      ProcessValue <- "UDT_Objetos_Valvulas_VM-52_estado"
   Button "Button_5" at 357,163 size 85x39; TextOff 'PERMEADO'
      on Click: ActivateScreen("4Permeado", 0)
   Button "Button_4" at 264,163 size 85x39; TextOff 'OSMOSIS'
      on Click: ActivateScreen("4Permeado", 0)
   IOField "I/O field_2" at 412,264 size 59x19; FormatPattern 9999; Unit  Bar
      ProcessValue <- "UDT_Objetos_Presion_PT-11_presion"
   IOField "I/O field_1" at 474,263 size 71x19; FormatPattern 9999; Unit  m3/h
      ProcessValue <- "UDT_Objetos_Flujo_FI-10_flujo"
   Bar "Bar_1" at 622,277 size 14x131; MinimumValue 0; MaximumValue 100
      ProcessValue <- "UDT_Objetos_Nivel_PT-13_nivel_porcentaje"
   IOField "I/O field_3" at 558,327 size 58x19; FormatPattern 9999; Unit  m3
      ProcessValue <- "UDT_Objetos_Nivel_PT-13_nivel_volumen"
   IOField "I/O field_4" at 572,347 size 44x19; FormatPattern 999; Unit  m
      ProcessValue <- "UDT_Objetos_Nivel_PT-13_nivel"

Template "Template_2" 800x480
   Button "Template_Button_5" at 200,440 size 99x39; TextOff 'ORP'
      on Click: ActivateScreen("ORP", 0)
   Button "Template_Button_6" at 100,440 size 99x39; TextOff 'CT'
      on Click: ActivateScreen("CT", 0)
   Button "Template_Button_7" at 0,440 size 99x39; TextOff 'COT'
      on Click: ActivateScreen("COT", 0)
   Button "Template_Button_3" at 400,440 size 99x39; TextOff 'TRB'
      on Click: ActivateScreen("TRB", 0)
   Button "Template_Button_4" at 300,440 size 99x39; TextOff 'PH'
      on Click: ActivateScreen("PH", 0)
   Button "Template_Button_1" at 500,441 size 99x39; TextOff 'FI'
      on Click: ActivateScreen("FI", 0)
   Button "Template_Button_2" at 600,441 size 99x39; TextOff 'RAD'
      on Click: ActivateScreen("RAD", 0)
   Button "Template_Button_8" at 700,441 size 99x39; TextOff 'PT'
      on Click: ActivateScreen("PT", 0)
   GraphicView "Graphic view_1" at 344,0 size 112x56; Picture "Coca-Cola_Femsa_Logo"
   Button "Template_Button_9" at 0,0 size 99x39; TextOff 'INICIO'
      on Click: ActivateScreen("0Ultrafiltracion", 0)

screen "Configuraciones" 800x480, template "Template_3"
   IOField "I/O field_1" at 51,95 size 96x32; FormatPattern s99999; Unit  Hz
      ProcessValue <- "UDT_Objetos_Bombas_BC-11_frecuencia"
   TextField "Text field_1" at 75,36 size 43x20; Text 'BC-11'
   TextField "Text field_3" at 60,57 size 74x36; Text 'Frecuencia Trabajo'
   IOField "I/O field_3" at 49,241 size 96x32; FormatPattern 999; Unit  mg/L
      ProcessValue <- "UDT_Objetos_Sensores_Especiales_COT-01_operacion_bajo"
   TextField "Text field_4" at 71,180 size 51x20; Text 'COT-01'
   TextField "Text field_5" at 40,202 size 114x36; Text 'Rango operación bajo'
   IOField "I/O field_4" at 49,314 size 96x32; FormatPattern 999; Unit  mg/L
      ProcessValue <- "UDT_Objetos_Sensores_Especiales_COT-01_operacion_alto"
   TextField "Text field_6" at 40,275 size 114x36; Text 'Rango operación alto'
   IOField "I/O field_5" at 49,387 size 96x32; FormatPattern 999; Unit  mg/L
      ProcessValue <- "UDT_Objetos_Sensores_Especiales_COT-01_trabajo_alto"
   TextField "Text field_7" at 63,348 size 67x36; Text 'Punto de trabajo'
   IOField "I/O field_6" at 219,240 size 96x32; FormatPattern 9999; Unit  mS
      ProcessValue <- "UDT_Objetos_Sensores_Especiales_CT-02_operacion_bajo"
   TextField "Text field_8" at 313,179 size 42x20; Text 'CT-02'
   TextField "Text field_9" at 210,201 size 114x36; Text 'Rango operación bajo'
   IOField "I/O field_7" at 219,313 size 96x32; FormatPattern 9999; Unit  mS
      ProcessValue <- "UDT_Objetos_Sensores_Especiales_CT-02_operacion_alto"
   TextField "Text field_10" at 210,274 size 114x36; Text 'Rango operación alto'
   IOField "I/O field_8" at 219,386 size 96x32; FormatPattern 9999; Unit  mS
      ProcessValue <- "UDT_Objetos_Sensores_Especiales_CT-02_trabajo_alto"
   TextField "Text field_11" at 226,347 size 82x36; Text 'Punto de trabajo alto'
   IOField "I/O field_9" at 349,240 size 96x32; FormatPattern 999; Unit  mS
      ProcessValue <- "UDT_Objetos_Sensores_Especiales_CT-02_trabajo_bajo"
   TextField "Text field_12" at 356,201 size 85x36; Text 'Punto de trabajo bajo'
   IOField "I/O field_2" at 523,240 size 96x32; FormatPattern s9999; Unit  mV
      ProcessValue <- "UDT_Objetos_Sensores_Especiales_ORP-01_operacion_bajo"
   TextField "Text field_2" at 611,179 size 53x20; Text 'ORP-01'
   TextField "Text field_13" at 514,201 size 114x36; Text 'Rango operación bajo'
   IOField "I/O field_10" at 523,313 size 96x32; FormatPattern s9999; Unit  mV
      ProcessValue <- "UDT_Objetos_Sensores_Especiales_ORP-01_operacion_alto"
   TextField "Text field_14" at 514,274 size 114x36; Text 'Rango operación alto'
   IOField "I/O field_11" at 523,386 size 96x32; FormatPattern s9999; Unit  mV
      ProcessValue <- "UDT_Objetos_Sensores_Especiales_ORP-01_trabajo_alto"
   TextField "Text field_15" at 530,347 size 82x36; Text 'Punto de trabajo alto'
   IOField "I/O field_12" at 653,240 size 96x32; FormatPattern s9999; Unit  mV
      ProcessValue <- "UDT_Objetos_Sensores_Especiales_ORP-01_trabajo_bajo"
   TextField "Text field_16" at 660,201 size 85x36; Text 'Punto de trabajo bajo'
   IOField "I/O field_13" at 202,95 size 96x32; FormatPattern s99999; Unit  s
      ProcessValue <- "UDT_Objetos_Bombas_BC-11_frecuencia"
   TextField "Text field_17" at 218,36 size 59x20; Text 'Valvulas'
   TextField "Text field_18" at 211,57 size 74x36; Text 'Tiempo de Alarma'
   Group "Group" at 185,26 size 125x118
   Group "Group_4" at 34,26 size 125x118
   Group "Group_5" at 508,169 size 259x255
   Group "Group_6" at 204,169 size 259x255
   Group "Group_7" at 34,170 size 125x255
   IOField "I/O field_16" at 658,95 size 96x32; FormatPattern 999; Unit  m2
      ProcessValue <- "UDT_Objetos_Nivel_PT-13_area_tanque"
   TextField "Text field_23" at 648,36 size 112x20; Text 'Tanque TK-INOX'
   TextField "Text field_24" at 685,65 size 37x20; Text 'Area'
   IOField "I/O field_15" at 506,95 size 96x32; FormatPattern 999; Unit  m2
      ProcessValue <- "UDT_Objetos_Nivel_PT-12_area_tanque"
   TextField "Text field_21" at 516,36 size 72x36; Text 'Tanque TK-PER-01'
   TextField "Text field_22" at 533,73 size 37x20; Text 'Area'
   IOField "I/O field_14" at 354,95 size 96x32; FormatPattern 999; Unit  m2
      ProcessValue <- "UDT_Objetos_Nivel_RAD-04_area_tanque"
   TextField "Text field_19" at 351,36 size 97x20; Text 'Tanque TK-06'
   TextField "Text field_20" at 381,65 size 37x20; Text 'Area'
   Button "Template_Button_7" at 0,440 size 99x39; TextOff 'COT'; PictureOff "Left_Arrow"
      on Click: ActivateScreen("Presion2", 0)
   Button "Template_Button_8" at 700,441 size 99x39; TextOff 'PT'; PictureOff "Right_Arrow"
      on Click: ActivateScreen("Configuraciones_1", 0)

screen "Configuraciones_1" 800x480, template "Template_3"
   IOField "I/O field_3" at 49,241 size 96x32; FormatPattern 99; Unit  pH
      ProcessValue <- "UDT_Objetos_Sensores_Especiales_PH-04_operacion_bajo"
   TextField "Text field_4" at 75,180 size 44x20; Text 'PH-04'
   TextField "Text field_5" at 40,202 size 114x36; Text 'Rango operación bajo'
   IOField "I/O field_4" at 49,314 size 96x32; FormatPattern 999; Unit  pH
      ProcessValue <- "UDT_Objetos_Sensores_Especiales_PH-04_operacion_bajo"
   TextField "Text field_6" at 40,275 size 114x36; Text 'Rango operación alto'
   IOField "I/O field_6" at 201,240 size 96x32; FormatPattern s9999; Unit  mV
      ProcessValue <- "UDT_Objetos_Sensores_Especiales_ORP-02_operacion_bajo"
   TextField "Text field_8" at 289,179 size 53x20; Text 'ORP-02'
   TextField "Text field_9" at 192,201 size 114x36; Text 'Rango operación bajo'
   IOField "I/O field_7" at 201,313 size 96x32; FormatPattern s9999; Unit  mV
      ProcessValue <- "UDT_Objetos_Sensores_Especiales_ORP-02_operacion_alto"
   TextField "Text field_10" at 192,274 size 114x36; Text 'Rango operación alto'
   IOField "I/O field_8" at 201,386 size 96x32; FormatPattern s9999; Unit  mV
      ProcessValue <- "UDT_Objetos_Sensores_Especiales_ORP-02_trabajo_alto"
   TextField "Text field_11" at 208,347 size 82x36; Text 'Punto de trabajo alto'
   IOField "I/O field_9" at 331,240 size 96x32; FormatPattern s9999; Unit  mV
      ProcessValue <- "UDT_Objetos_Sensores_Especiales_ORP-02_trabajo_bajo"
   TextField "Text field_12" at 338,201 size 85x36; Text 'Punto de trabajo bajo'
   IOField "I/O field_2" at 484,240 size 96x32; FormatPattern s9999; Unit  NTU
      ProcessValue <- "UDT_Objetos_Sensores_Especiales_TRB-02_operacion_bajo"
   TextField "Text field_2" at 573,179 size 51x20; Text 'TRB-02'
   TextField "Text field_13" at 475,201 size 114x36; Text 'Rango operación bajo'
   IOField "I/O field_10" at 484,313 size 96x32; FormatPattern s9999; Unit  NTU
      ProcessValue <- "UDT_Objetos_Sensores_Especiales_TRB-02_operacion_alto"
   TextField "Text field_14" at 475,274 size 114x36; Text 'Rango operación alto'
   IOField "I/O field_11" at 484,386 size 96x32; FormatPattern s9999; Unit  NTU
      ProcessValue <- "UDT_Objetos_Sensores_Especiales_TRB-02_trabajo_alto"
   TextField "Text field_15" at 491,347 size 82x36; Text 'Punto de trabajo alto'
   IOField "I/O field_12" at 614,240 size 96x32; FormatPattern s9999; Unit  NTU
      ProcessValue <- "UDT_Objetos_Sensores_Especiales_TRB-02_trabajo_bajo"
   TextField "Text field_16" at 621,201 size 85x36; Text 'Punto de trabajo bajo'
   IOField "I/O field_14" at 51,95 size 96x32; FormatPattern 999; Unit  m2
      ProcessValue <- "UDT_Objetos_Nivel_PT-07_area_tanque"
   TextField "Text field_19" at 48,36 size 97x20; Text 'Tanque TK-03'
   TextField "Text field_20" at 78,65 size 37x20; Text 'Area'
   IOField "I/O field_1" at 202,95 size 96x32; FormatPattern 999; Unit  m2
      ProcessValue <- "UDT_Objetos_Nivel_RAD-06_area_tanque"
   TextField "Text field_1" at 216,36 size 64x20; Text 'Tanque 5'
   TextField "Text field_3" at 229,65 size 37x20; Text 'Area'
   IOField "I/O field_5" at 354,95 size 96x32; FormatPattern 999; Unit  m2
      ProcessValue <- "UDT_Objetos_Nivel_RAD-05_area_tanque"
   TextField "Text field_7" at 368,36 size 64x20; Text 'Tanque 4'
   TextField "Text field_17" at 381,65 size 37x20; Text 'Area'
   Button "Template_Button_7" at 0,440 size 99x39; TextOff 'COT'; PictureOff "Left_Arrow"
      on Click: ActivateScreen("Configuraciones", 0)
   Button "Template_Button_8" at 700,441 size 99x39; TextOff 'PT'; PictureOff "Right_Arrow"
      on Click: ActivateScreen("Configuraciones_2", 0)

screen "Configuraciones_2" 800x480, template "Template_3"
   IOField "I/O field_1" at 51,95 size 96x32; FormatPattern s99999
      ProcessValue <- "UDT_Objetos_Bombas_BC-11_frecuencia"
   TextField "Text field_1" at 75,36 size 32x20; Text 'XXX'
   TextField "Text field_3" at 60,57 size 74x36; Text 'Frecuencia Trabajo'
   IOField "I/O field_3" at 49,241 size 96x32; FormatPattern 999
      ProcessValue <- "UDT_Objetos_Sensores_Especiales_COT-01_operacion_bajo"
   TextField "Text field_4" at 81,180 size 32x20; Text 'XXX'
   TextField "Text field_5" at 40,202 size 114x36; Text 'Rango operación bajo'
   IOField "I/O field_4" at 49,314 size 96x32; FormatPattern 999
      ProcessValue <- "UDT_Objetos_Sensores_Especiales_COT-01_operacion_alto"
   TextField "Text field_6" at 40,275 size 114x36; Text 'Rango operación alto'
   IOField "I/O field_5" at 49,387 size 96x32; FormatPattern 999
      ProcessValue <- "UDT_Objetos_Sensores_Especiales_COT-01_trabajo_alto"
   TextField "Text field_7" at 63,348 size 67x36; Text 'Punto de trabajo'
   IOField "I/O field_6" at 201,240 size 96x32; FormatPattern 9999
      ProcessValue <- "UDT_Objetos_Flujo_FI-06_operacion_bajo"
   TextField "Text field_8" at 295,179 size 38x20; Text 'FI-06'
   TextField "Text field_9" at 192,201 size 114x36; Text 'Rango operación bajo'
   IOField "I/O field_7" at 201,313 size 96x32; FormatPattern 9999
      ProcessValue <- "UDT_Objetos_Flujo_FI-06_operacion_alto"
   TextField "Text field_10" at 192,274 size 114x36; Text 'Rango operación alto'
   IOField "I/O field_8" at 201,386 size 96x32; FormatPattern 9999
      ProcessValue <- "UDT_Objetos_Flujo_FI-06_trabajo_alto"
   TextField "Text field_11" at 208,347 size 82x36; Text 'Punto de trabajo alto'
   IOField "I/O field_9" at 331,240 size 96x32; FormatPattern 9999
      ProcessValue <- "UDT_Objetos_Flujo_FI-06_trabajo_bajo"
   TextField "Text field_12" at 338,201 size 85x36; Text 'Punto de trabajo bajo'
   IOField "I/O field_2" at 484,240 size 96x32; FormatPattern s9999
      ProcessValue <- "UDT_Objetos_Flujo_FI-07_operacion_bajo"
   TextField "Text field_2" at 572,179 size 38x20; Text 'FI-07'
   TextField "Text field_13" at 475,201 size 114x36; Text 'Rango operación bajo'
   IOField "I/O field_10" at 484,313 size 96x32; FormatPattern s9999
      ProcessValue <- "UDT_Objetos_Flujo_FI-07_operacion_alto"
   TextField "Text field_14" at 475,274 size 114x36; Text 'Rango operación alto'
   IOField "I/O field_11" at 484,386 size 96x32; FormatPattern s9999
      ProcessValue <- "UDT_Objetos_Flujo_FI-07_trabajo_alto"
   TextField "Text field_15" at 491,347 size 82x36; Text 'Punto de trabajo alto'
   IOField "I/O field_12" at 614,240 size 96x32; FormatPattern s9999
      ProcessValue <- "UDT_Objetos_Flujo_FI-07_trabajo_bajo"
   TextField "Text field_16" at 621,201 size 85x36; Text 'Punto de trabajo bajo'
   Button "Template_Button_7" at 0,440 size 99x39; TextOff 'COT'; PictureOff "Left_Arrow"
      on Click: ActivateScreen("Configuraciones_1", 0)
   Button "Template_Button_8" at 700,441 size 99x39; TextOff 'PT'; PictureOff "Right_Arrow"
      on Click: ActivateScreen("Configuraciones_3", 0)

